LIN {X 0,Y 254.64,Z 783.41,A -85,B 0,C 180,E1 -18457.933,E2 -18457.933} C_VEL
LIN {X 0,Y 255.196,Z 782.528,A -85,B 0,C 180,E1 -18459.512,E2 -18459.512} C_VEL
LIN {X 0,Y 255.928,Z 781.105,A -85,B 0,C 180,E1 -18461.084,E2 -18461.084} C_VEL
LIN {X 0,Y 257.325,Z 777.923,A -85,B 0,C 180,E1 -18463.425,E2 -18463.425} C_VEL
LIN {X 0,Y 259.009,Z 773.292,A -85,B 0,C 180,E1 -18465.745,E2 -18465.745} C_VEL
LIN {X 0,Y 260.929,Z 768.168,A -85,B 0,C 180,E1 -18467.64,E2 -18467.64} C_VEL
LIN {X 0,Y 262.981,Z 761.785,A -85,B 0,C 180,E1 -18469.516,E2 -18469.516} C_VEL
LIN {X 0,Y 265.315,Z 753.655,A -85,B 0,C 180,E1 -18471.407,E2 -18471.407} C_VEL
LIN {X 0,Y 267.313,Z 745.611,A -85,B 0,C 180,E1 -18472.889,E2 -18472.889} C_VEL
LIN {X 0,Y 269.342,Z 736.316,A -85,B 0,C 180,E1 -18474.267,E2 -18474.267} C_VEL
LIN {X 0,Y 271.322,Z 725.43,A -85,B 0,C 180,E1 -18475.509,E2 -18475.509} C_VEL
LIN {X 0,Y 272.904,Z 714.301,A -85,B 0,C 180,E1 -18476.479,E2 -18476.479} C_VEL
LIN {X 0,Y 274.215,Z 699.395,A -85,B 0,C 180,E1 -18477.423,E2 -18477.423} C_VEL
LIN {X 0,Y 278.601,Z 663.75,A -85,B 0,C 180,E1 -18479.26,E2 -18479.26} C_VEL
LIN {X 0,Y 282.632,Z 634.038,A -85,B 0,C 180,E1 -18480.701,E2 -18480.701} C_VEL
LIN {X 0,Y 282.883,Z 631.989,A -85,B 0,C 180,E1 -18480.826,E2 -18480.826} C_VEL
LIN {X 0,Y 286.551,Z 622.135,A -85,B 0,C 180,E1 -18481.825,E2 -18481.825} C_VEL
LIN {X 0,Y 289.01,Z 614.087,A -85,B 0,C 180,E1 -18483.007,E2 -18483.007} C_VEL
LIN {X 0,Y 289.054,Z 610.102,A -85,B 0,C 180,E1 -18484.242,E2 -18484.242} C_VEL
LIN {X 0,Y 288.786,Z 608.298,A -85,B 0,C 180,E1 -18485.033,E2 -18485.033} C_VEL
LIN {X 0,Y 287.847,Z 606.637,A -85,B 0,C 180,E1 -18486.32,E2 -18486.32} C_VEL
LIN {X 0,Y 286.56,Z 604.936,A -85,B 0,C 180,E1 -18488.296,E2 -18488.296} C_VEL
LIN {X 0,Y 285.583,Z 604.023,A -85,B 0,C 180,E1 -18490.28,E2 -18490.28} C_VEL
LIN {X 0,Y 284.947,Z 603.772,A -85,B 0,C 180,E1 -18492.275,E2 -18492.275} C_VEL
LIN {X 0,Y 284.613,Z 604.193,A -85,B 0,C 180,E1 -18494.266,E2 -18494.266} C_VEL
LIN {X 0,Y 284.469,Z 605.335,A -85,B 0,C 180,E1 -18496.23,E2 -18496.23} C_VEL
LIN {X 0,Y 284.524,Z 608.104,A -85,B 0,C 180,E1 -18498.967,E2 -18498.967} C_VEL
LIN {X 0,Y 284.591,Z 611.178,A -85,B 0,C 180,E1 -18501.037,E2 -18501.037} C_VEL
LIN {X 0,Y 284.604,Z 615.38,A -85,B 0,C 180,E1 -18503.209,E2 -18503.209} C_VEL
LIN {X 0,Y 284.52,Z 617.632,A -85,B 0,C 180,E1 -18504.2,E2 -18504.2} C_VEL
LIN {X 0,Y 283.942,Z 619.835,A -85,B 0,C 180,E1 -18504.867,E2 -18504.867} C_VEL
LIN {X 0,Y 279.716,Z 632.839,A -85,B 0,C 180,E1 -18508.101,E2 -18508.101} C_VEL
LIN {X 0,Y 281.369,Z 646.293,A -85,B 0,C 180,E1 -18509.997,E2 -18509.997} C_VEL
LIN {X 0,Y 282.942,Z 661.375,A -85,B 0,C 180,E1 -18511.756,E2 -18511.756} C_VEL
LIN {X 0,Y 283.284,Z 668.767,A -85,B 0,C 180,E1 -18512.455,E2 -18512.455} C_VEL
LIN {X 0,Y 278.495,Z 708.238,A -85,B 0,C 180,E1 -18514.295,E2 -18514.295} C_VEL
LIN {X 0,Y 276.699,Z 719.034,A -85,B 0,C 180,E1 -18515.022,E2 -18515.022} C_VEL
LIN {X 0,Y 274.44,Z 729.554,A -85,B 0,C 180,E1 -18516.013,E2 -18516.013} C_VEL
LIN {X 0,Y 272.006,Z 739.288,A -85,B 0,C 180,E1 -18517.197,E2 -18517.197} C_VEL
LIN {X 0,Y 269.353,Z 748.071,A -85,B 0,C 180,E1 -18518.575,E2 -18518.575} C_VEL
LIN {X 0,Y 267,Z 755.114,A -85,B 0,C 180,E1 -18519.99,E2 -18519.99} C_VEL
LIN {X 0,Y 264.343,Z 762.314,A -85,B 0,C 180,E1 -18521.796,E2 -18521.796} C_VEL
LIN {X 0,Y 261.944,Z 768.017,A -85,B 0,C 180,E1 -18523.637,E2 -18523.637} C_VEL
LIN {X 0,Y 259.412,Z 773.188,A -85,B 0,C 180,E1 -18525.887,E2 -18525.887} C_VEL
LIN {X 0,Y 258.13,Z 775.765,A -85,B 0,C 180,E1 -18527.419,E2 -18527.419} C_VEL
LIN {X 0,Y 257.031,Z 777.741,A -85,B 0,C 180,E1 -18528.965,E2 -18528.965} C_VEL
LIN {X 0,Y 256.07,Z 779.154,A -85,B 0,C 180,E1 -18530.522,E2 -18530.522} C_VEL
LIN {X 0,Y 255.228,Z 780.071,A -85,B 0,C 180,E1 -18532.445,E2 -18532.445} C_VEL
LIN {X 0,Y 254.805,Z 780.276,A -85,B 0,C 180,E1 -18533.666,E2 -18533.666} C_VEL
LIN {X 0,Y 254.337,Z 779.949,A -85,B 0,C 180,E1 -18535.245,E2 -18535.245} C_VEL
LIN {X 0,Y 254.123,Z 779.049,A -85,B 0,C 180,E1 -18536.829,E2 -18536.829} C_VEL
LIN {X 0,Y 254.003,Z 776.68,A -85,B 0,C 180,E1 -18539.207,E2 -18539.207} C_VEL
LIN {X 0,Y 254.05,Z 772.777,A -85,B 0,C 180,E1 -18541.585,E2 -18541.585} C_VEL
LIN {X 0,Y 254.225,Z 769.338,A -85,B 0,C 180,E1 -18543.17,E2 -18543.17} C_VEL
LIN {X 0,Y 254.358,Z 765.073,A -85,B 0,C 180,E1 -18544.755,E2 -18544.755} C_VEL
LIN {X 0,Y 254.634,Z 758.449,A -85,B 0,C 180,E1 -18546.737,E2 -18546.737} C_VEL
LIN {X 0,Y 254.986,Z 751.78,A -85,B 0,C 180,E1 -18548.32,E2 -18548.32} C_VEL
LIN {X 0,Y 255.449,Z 743.401,A -85,B 0,C 180,E1 -18549.901,E2 -18549.901} C_VEL
LIN {X 0,Y 255.9,Z 734.328,A -85,B 0,C 180,E1 -18551.285,E2 -18551.285} C_VEL
LIN {X 0,Y 256.485,Z 723.294,A -85,B 0,C 180,E1 -18552.562,E2 -18552.562} C_VEL
LIN {X 0,Y 256.869,Z 713.102,A -85,B 0,C 180,E1 -18553.448,E2 -18553.448} C_VEL
LIN {X 0,Y 257.314,Z 700.732,A -85,B 0,C 180,E1 -18554.18,E2 -18554.18} C_VEL
LIN {X 0,Y 258.285,Z 654.86,A -85,B 0,C 180,E1 -18556.218,E2 -18556.218} C_VEL
LIN {X 0,Y 256.91,Z 633.005,A -85,B 0,C 180,E1 -18557.211,E2 -18557.211} C_VEL
LIN {X 0,Y 256.915,Z 631.92,A -85,B 0,C 180,E1 -18557.311,E2 -18557.311} C_VEL
LIN {X 0,Y 258.388,Z 612.535,A -85,B 0,C 180,E1 -18561.543,E2 -18561.543} C_VEL
LIN {X 0,Y 259.975,Z 593.835,A -85,B 0,C 180,E1 -18565.629,E2 -18565.629} C_VEL
LIN {X 0,Y 261.374,Z 578.642,A -85,B 0,C 180,E1 -18568.947,E2 -18568.947} C_VEL
LIN {X 0,Y 260.158,Z 571.5,A -85,B 0,C 180,E1 -18570.601,E2 -18570.601} C_VEL
LIN {X 0,Y 256.188,Z 552.77,A -85,B 0,C 180,E1 -18575.125,E2 -18575.125} C_VEL
LIN {X 0,Y 256.077,Z 552.583,A -85,B 0,C 180,E1 -18579.141,E2 -18579.141} C_VEL
LIN {X 0,Y 256.07,Z 552.534,A -85,B 0,C 180,E1 -18583.326,E2 -18583.326} C_VEL
LIN {X 0,Y 256.093,Z 552.578,A -85,B 0,C 180,E1 -18587.814,E2 -18587.814} C_VEL
LIN {X 0,Y 256.078,Z 552.55,A -85,B 0,C 180,E1 -18590.858,E2 -18590.858} C_VEL
LIN {X 0,Y 256.134,Z 552.571,A -85,B 0,C 180,E1 -18592.867,E2 -18592.867} C_VEL
LIN {X 0,Y 256.153,Z 552.697,A -85,B 0,C 180,E1 -18596.5,E2 -18596.5} C_VEL
LIN {X 0,Y 256.89,Z 555.634,A -85,B 0,C 180,E1 -18597.795,E2 -18597.795} C_VEL
LIN {X 0,Y 264.799,Z 571.908,A -85,B 0,C 180,E1 -18599.433,E2 -18599.433} C_VEL
LIN {X 0,Y 271.817,Z 588.537,A -85,B 0,C 180,E1 -18600.806,E2 -18600.806} C_VEL
LIN {X 0,Y 273.608,Z 593.478,A -85,B 0,C 180,E1 -18601.163,E2 -18601.163} C_VEL
LIN {X 0,Y 271.526,Z 660.332,A -85,B 0,C 180,E1 -18602.909,E2 -18602.909} C_VEL
LIN {X 0,Y 270.584,Z 673.573,A -85,B 0,C 180,E1 -18603.485,E2 -18603.485} C_VEL
LIN {X 0,Y 269.339,Z 686.707,A -85,B 0,C 180,E1 -18604.393,E2 -18604.393} C_VEL
LIN {X 0,Y 267.637,Z 699.141,A -85,B 0,C 180,E1 -18605.568,E2 -18605.568} C_VEL
LIN {X 0,Y 265.652,Z 710.78,A -85,B 0,C 180,E1 -18607.03,E2 -18607.03} C_VEL
LIN {X 0,Y 263.919,Z 719.999,A -85,B 0,C 180,E1 -18608.488,E2 -18608.488} C_VEL
LIN {X 0,Y 262.043,Z 729.759,A -85,B 0,C 180,E1 -18610.411,E2 -18610.411} C_VEL
LIN {X 0,Y 260.236,Z 737.623,A -85,B 0,C 180,E1 -18612.311,E2 -18612.311} C_VEL
LIN {X 0,Y 258.368,Z 745.305,A -85,B 0,C 180,E1 -18614.619,E2 -18614.619} C_VEL
LIN {X 0,Y 256.723,Z 752.357,A -85,B 0,C 180,E1 -18617.348,E2 -18617.348} C_VEL
LIN {X 0,Y 255.59,Z 757.052,A -85,B 0,C 180,E1 -18619.703,E2 -18619.703} C_VEL
LIN {X 0,Y 254.885,Z 760.637,A -85,B 0,C 180,E1 -18622.074,E2 -18622.074} C_VEL
LIN {X 0,Y 254.515,Z 762.597,A -85,B 0,C 180,E1 -18623.765,E2 -18623.765} C_VEL
LIN {X 0,Y 254.194,Z 764.873,A -85,B 0,C 180,E1 -18626.829,E2 -18626.829} C_VEL
LIN {X 0,Y 254.096,Z 765.484,A -85,B 0,C 180,E1 -18628.414,E2 -18628.414} C_VEL
LIN {X 0,Y 254.064,Z 765.714,A -85,B 0,C 180,E1 -18629.999,E2 -18629.999} C_VEL
LIN {X 0,Y 254.095,Z 765.522,A -85,B 0,C 180,E1 -18631.584,E2 -18631.584} C_VEL
LIN {X 0,Y 254.192,Z 764.937,A -85,B 0,C 180,E1 -18633.168,E2 -18633.168} C_VEL
LIN {X 0,Y 254.534,Z 762.617,A -85,B 0,C 180,E1 -18636.339,E2 -18636.339} C_VEL
LIN {X 0,Y 255.077,Z 759.749,A -85,B 0,C 180,E1 -18638.715,E2 -18638.715} C_VEL
LIN {X 0,Y 255.91,Z 755.858,A -85,B 0,C 180,E1 -18641.082,E2 -18641.082} C_VEL
LIN {X 0,Y 257.1,Z 750.84,A -85,B 0,C 180,E1 -18643.434,E2 -18643.434} C_VEL
LIN {X 0,Y 258.531,Z 744.522,A -85,B 0,C 180,E1 -18645.772,E2 -18645.772} C_VEL
LIN {X 0,Y 260.488,Z 736.605,A -85,B 0,C 180,E1 -18648.074,E2 -18648.074} C_VEL
LIN {X 0,Y 262.351,Z 728.536,A -85,B 0,C 180,E1 -18649.97,E2 -18649.97} C_VEL
LIN {X 0,Y 264.206,Z 718.694,A -85,B 0,C 180,E1 -18651.862,E2 -18651.862} C_VEL
LIN {X 0,Y 266.253,Z 707.61,A -85,B 0,C 180,E1 -18653.529,E2 -18653.529} C_VEL
LIN {X 0,Y 268.044,Z 696.735,A -85,B 0,C 180,E1 -18654.802,E2 -18654.802} C_VEL
LIN {X 0,Y 269.616,Z 684.708,A -85,B 0,C 180,E1 -18655.887,E2 -18655.887} C_VEL
LIN {X 0,Y 270.803,Z 672.349,A -85,B 0,C 180,E1 -18656.697,E2 -18656.697} C_VEL
LIN {X 0,Y 271.68,Z 659.521,A -85,B 0,C 180,E1 -18657.228,E2 -18657.228} C_VEL
LIN {X 0,Y 273.728,Z 593.612,A -85,B 0,C 180,E1 -18658.945,E2 -18658.945} C_VEL
LIN {X 0,Y 266.65,Z 575.933,A -85,B 0,C 180,E1 -18660.336,E2 -18660.336} C_VEL
LIN {X 0,Y 258.473,Z 559.011,A -85,B 0,C 180,E1 -18661.953,E2 -18661.953} C_VEL
LIN {X 0,Y 256.796,Z 555.428,A -85,B 0,C 180,E1 -18662.39,E2 -18662.39} C_VEL
LIN {X 0,Y 256.138,Z 552.622,A -85,B 0,C 180,E1 -18663.719,E2 -18663.719} C_VEL
LIN {X 0,Y 256.127,Z 552.578,A -85,B 0,C 180,E1 -18667.274,E2 -18667.274} C_VEL
LIN {X 0,Y 256.053,Z 552.584,A -85,B 0,C 180,E1 -18671.201,E2 -18671.201} C_VEL
LIN {X 0,Y 256.057,Z 552.569,A -85,B 0,C 180,E1 -18675.528,E2 -18675.528} C_VEL
LIN {X 0,Y 256.079,Z 552.582,A -85,B 0,C 180,E1 -18678.801,E2 -18678.801} C_VEL
LIN {X 0,Y 256.149,Z 552.557,A -85,B 0,C 180,E1 -18682.87,E2 -18682.87} C_VEL
LIN {X 0,Y 256.08,Z 552.582,A -85,B 0,C 180,E1 -18686.709,E2 -18686.709} C_VEL
LIN {X 0,Y 256.132,Z 552.572,A -85,B 0,C 180,E1 -18691.404,E2 -18691.404} C_VEL
LIN {X 0,Y 256.149,Z 552.574,A -85,B 0,C 180,E1 -18695.822,E2 -18695.822} C_VEL
LIN {X 0,Y 256.16,Z 552.567,A -85,B 0,C 180,E1 -18699.104,E2 -18699.104} C_VEL
LIN {X 0,Y 256.208,Z 552.56,A -85,B 0,C 180,E1 -18702.664,E2 -18702.664} C_VEL
LIN {X 0,Y 255.561,Z 552.637,A -85,B 0,C 180,E1 -18703.976,E2 -18703.976} C_VEL
LIN {X 0,Y 252.702,Z 553.006,A -85,B 0,C 180,E1 -18706.116,E2 -18706.116} C_VEL
LIN {X 0,Y 250.308,Z 553.301,A -85,B 0,C 180,E1 -18707.859,E2 -18707.859} C_VEL
LIN {X 0,Y 249.349,Z 553.411,A -85,B 0,C 180,E1 -18709.21,E2 -18709.21} C_VEL
LIN {X 0,Y 249.309,Z 553.412,A -85,B 0,C 180,E1 -18709.667,E2 -18709.667} C_VEL
LIN {X 0,Y 249.475,Z 553.401,A -85,B 0,C 180,E1 -18711.903,E2 -18711.903} C_VEL
LIN {X 0,Y 249.43,Z 553.396,A -85,B 0,C 180,E1 -18716.769,E2 -18716.769} C_VEL
LIN {X 0,Y 249.729,Z 553.378,A -85,B 0,C 180,E1 -18720,E2 -18720} C_VEL
LIN {X 0,Y 249.43,Z 553.398,A -85,B 0,C 180,E1 -18723.23,E2 -18723.23} C_VEL
LIN {X 0,Y 249.478,Z 553.404,A -85,B 0,C 180,E1 -18728.097,E2 -18728.097} C_VEL
LIN {X 0,Y 249.246,Z 553.426,A -85,B 0,C 180,E1 -18731.384,E2 -18731.384} C_VEL
LIN {X 0,Y 249.235,Z 553.424,A -85,B 0,C 180,E1 -18736.379,E2 -18736.379} C_VEL
LIN {X 0,Y 249.081,Z 553.447,A -85,B 0,C 180,E1 -18741.519,E2 -18741.519} C_VEL
LIN {X 0,Y 249.123,Z 553.448,A -85,B 0,C 180,E1 -18745.482,E2 -18745.482} C_VEL
LIN {X 0,Y 249.066,Z 553.461,A -85,B 0,C 180,E1 -18748.99,E2 -18748.99} C_VEL
LIN {X 0,Y 249.024,Z 553.465,A -85,B 0,C 180,E1 -18752.427,E2 -18752.427} C_VEL
LIN {X 0,Y 249.024,Z 553.436,A -85,B 0,C 180,E1 -18756.346,E2 -18756.346} C_VEL
LIN {X 0,Y 249.03,Z 553.464,A -85,B 0,C 180,E1 -18760.473,E2 -18760.473} C_VEL
LIN {X 0,Y 249.015,Z 553.468,A -85,B 0,C 180,E1 -18764.877,E2 -18764.877} C_VEL
LIN {X 0,Y 249.077,Z 553.446,A -85,B 0,C 180,E1 -18767.378,E2 -18767.378} C_VEL
LIN {X 0,Y 249.119,Z 553.651,A -85,B 0,C 180,E1 -18771.056,E2 -18771.056} C_VEL
LIN {X 0,Y 250.889,Z 560.889,A -85,B 0,C 180,E1 -18774.327,E2 -18774.327} C_VEL
LIN {X 0,Y 252.417,Z 567.594,A -85,B 0,C 180,E1 -18777.053,E2 -18777.053} C_VEL
LIN {X 0,Y 258.204,Z 580.32,A -85,B 0,C 180,E1 -18778.332,E2 -18778.332} C_VEL
LIN {X 0,Y 263,Z 592.075,A -85,B 0,C 180,E1 -18779.336,E2 -18779.336} C_VEL
LIN {X 0,Y 266.778,Z 617.218,A -85,B 0,C 180,E1 -18780.575,E2 -18780.575} C_VEL
LIN {X 0,Y 264.813,Z 676.163,A -85,B 0,C 180,E1 -18782.167,E2 -18782.167} C_VEL
LIN {X 0,Y 263.611,Z 690.053,A -85,B 0,C 180,E1 -18782.836,E2 -18782.836} C_VEL
LIN {X 0,Y 262.061,Z 702.494,A -85,B 0,C 180,E1 -18783.738,E2 -18783.738} C_VEL
LIN {X 0,Y 260.345,Z 713.602,A -85,B 0,C 180,E1 -18784.84,E2 -18784.84} C_VEL
LIN {X 0,Y 258.166,Z 725.168,A -85,B 0,C 180,E1 -18786.327,E2 -18786.327} C_VEL
LIN {X 0,Y 255.993,Z 735.585,A -85,B 0,C 180,E1 -18788.036,E2 -18788.036} C_VEL
LIN {X 0,Y 254.117,Z 744.109,A -85,B 0,C 180,E1 -18789.777,E2 -18789.777} C_VEL
LIN {X 0,Y 252.362,Z 752.159,A -85,B 0,C 180,E1 -18791.797,E2 -18791.797} C_VEL
LIN {X 0,Y 250.528,Z 759.66,A -85,B 0,C 180,E1 -18794.128,E2 -18794.128} C_VEL
LIN {X 0,Y 248.79,Z 766.747,A -85,B 0,C 180,E1 -18796.94,E2 -18796.94} C_VEL
LIN {X 0,Y 247.858,Z 771.468,A -85,B 0,C 180,E1 -18799.381,E2 -18799.381} C_VEL
LIN {X 0,Y 247.267,Z 775.082,A -85,B 0,C 180,E1 -18801.831,E2 -18801.831} C_VEL
LIN {X 0,Y 247.009,Z 776.944,A -85,B 0,C 180,E1 -18803.467,E2 -18803.467} C_VEL
LIN {X 0,Y 246.882,Z 778.341,A -85,B 0,C 180,E1 -18805.102,E2 -18805.102} C_VEL
LIN {X 0,Y 246.865,Z 779.339,A -85,B 0,C 180,E1 -18806.737,E2 -18806.737} C_VEL
LIN {X 0,Y 246.923,Z 779.949,A -85,B 0,C 180,E1 -18808.37,E2 -18808.37} C_VEL
LIN {X 0,Y 246.949,Z 780.095,A -85,B 0,C 180,E1 -18811.225,E2 -18811.225} C_VEL
LIN {X 0,Y 246.947,Z 782.169,A -85,B 0,C 180,E1 -18813.264,E2 -18813.264} C_VEL
LIN {X 0,Y 247.047,Z 783.354,A -85,B 0,C 180,E1 -18815.325,E2 -18815.325} C_VEL
LIN {X 0,Y 247.614,Z 783.463,A -85,B 0,C 180,E1 -18818.16,E2 -18818.16} C_VEL
LIN {X 0,Y 248.201,Z 782.811,A -85,B 0,C 180,E1 -18819.783,E2 -18819.783} C_VEL
LIN {X 0,Y 248.985,Z 781.614,A -85,B 0,C 180,E1 -18821.397,E2 -18821.397} C_VEL
LIN {X 0,Y 250.463,Z 778.708,A -85,B 0,C 180,E1 -18823.8,E2 -18823.8} C_VEL
LIN {X 0,Y 252.303,Z 774.521,A -85,B 0,C 180,E1 -18826.175,E2 -18826.175} C_VEL
LIN {X 0,Y 254.75,Z 768.662,A -85,B 0,C 180,E1 -18828.499,E2 -18828.499} C_VEL
LIN {X 0,Y 257.017,Z 762.49,A -85,B 0,C 180,E1 -18830.406,E2 -18830.406} C_VEL
LIN {X 0,Y 259.535,Z 754.826,A -85,B 0,C 180,E1 -18832.28,E2 -18832.28} C_VEL
LIN {X 0,Y 262.002,Z 746.136,A -85,B 0,C 180,E1 -18833.938,E2 -18833.938} C_VEL
LIN {X 0,Y 264.356,Z 736.691,A -85,B 0,C 180,E1 -18835.386,E2 -18835.386} C_VEL
LIN {X 0,Y 266.514,Z 725.928,A -85,B 0,C 180,E1 -18836.635,E2 -18836.635} C_VEL
LIN {X 0,Y 268.425,Z 714.14,A -85,B 0,C 180,E1 -18837.694,E2 -18837.694} C_VEL
LIN {X 0,Y 270.241,Z 697.254,A -85,B 0,C 180,E1 -18838.76,E2 -18838.76} C_VEL
LIN {X 0,Y 274.782,Z 663.805,A -85,B 0,C 180,E1 -18840.501,E2 -18840.501} C_VEL
LIN {X 0,Y 279.106,Z 634.046,A -85,B 0,C 180,E1 -18841.978,E2 -18841.978} C_VEL
LIN {X 0,Y 279.349,Z 632.11,A -85,B 0,C 180,E1 -18842.106,E2 -18842.106} C_VEL
LIN {X 0,Y 282.562,Z 623.941,A -85,B 0,C 180,E1 -18842.963,E2 -18842.963} C_VEL
LIN {X 0,Y 284.56,Z 618.001,A -85,B 0,C 180,E1 -18843.841,E2 -18843.841} C_VEL
LIN {X 0,Y 284.694,Z 615.564,A -85,B 0,C 180,E1 -18844.597,E2 -18844.597} C_VEL
LIN {X 0,Y 284.501,Z 613.728,A -85,B 0,C 180,E1 -18845.393,E2 -18845.393} C_VEL
LIN {X 0,Y 283.058,Z 611.491,A -85,B 0,C 180,E1 -18847.39,E2 -18847.39} C_VEL
LIN {X 0,Y 281.903,Z 610.195,A -85,B 0,C 180,E1 -18849.39,E2 -18849.39} C_VEL
LIN {X 0,Y 281.036,Z 609.577,A -85,B 0,C 180,E1 -18851.39,E2 -18851.39} C_VEL
LIN {X 0,Y 280.49,Z 609.675,A -85,B 0,C 180,E1 -18853.395,E2 -18853.395} C_VEL
LIN {X 0,Y 280.182,Z 610.456,A -85,B 0,C 180,E1 -18855.385,E2 -18855.385} C_VEL
LIN {X 0,Y 280.014,Z 611.963,A -85,B 0,C 180,E1 -18857.338,E2 -18857.338} C_VEL
LIN {X 0,Y 279.951,Z 614.125,A -85,B 0,C 180,E1 -18859.253,E2 -18859.253} C_VEL
LIN {X 0,Y 279.836,Z 618.383,A -85,B 0,C 180,E1 -18861.924,E2 -18861.924} C_VEL
LIN {X 0,Y 279.619,Z 621.758,A -85,B 0,C 180,E1 -18863.544,E2 -18863.544} C_VEL
LIN {X 0,Y 278.918,Z 624.069,A -85,B 0,C 180,E1 -18864.26,E2 -18864.26} C_VEL
LIN {X 0,Y 275.821,Z 633.078,A -85,B 0,C 180,E1 -18866.523,E2 -18866.523} C_VEL
LIN {X 0,Y 277.151,Z 646.617,A -85,B 0,C 180,E1 -18868.591,E2 -18868.591} C_VEL
LIN {X 0,Y 278.438,Z 661.312,A -85,B 0,C 180,E1 -18870.437,E2 -18870.437} C_VEL
LIN {X 0,Y 278.893,Z 670.399,A -85,B 0,C 180,E1 -18871.362,E2 -18871.362} C_VEL
LIN {X 0,Y 273.775,Z 708.71,A -85,B 0,C 180,E1 -18873.202,E2 -18873.202} C_VEL
LIN {X 0,Y 271.883,Z 719.441,A -85,B 0,C 180,E1 -18873.932,E2 -18873.932} C_VEL
LIN {X 0,Y 269.494,Z 729.878,A -85,B 0,C 180,E1 -18874.927,E2 -18874.927} C_VEL
LIN {X 0,Y 266.898,Z 739.436,A -85,B 0,C 180,E1 -18876.118,E2 -18876.118} C_VEL
LIN {X 0,Y 263.7,Z 749.041,A -85,B 0,C 180,E1 -18877.68,E2 -18877.68} C_VEL
LIN {X 0,Y 261.19,Z 755.969,A -85,B 0,C 180,E1 -18879.113,E2 -18879.113} C_VEL
LIN {X 0,Y 258.353,Z 763.027,A -85,B 0,C 180,E1 -18880.947,E2 -18880.947} C_VEL
LIN {X 0,Y 256.218,Z 767.56,A -85,B 0,C 180,E1 -18882.439,E2 -18882.439} C_VEL
LIN {X 0,Y 253.458,Z 772.814,A -85,B 0,C 180,E1 -18884.727,E2 -18884.727} C_VEL
LIN {X 0,Y 251.953,Z 775.512,A -85,B 0,C 180,E1 -18886.285,E2 -18886.285} C_VEL
LIN {X 0,Y 250.12,Z 778.385,A -85,B 0,C 180,E1 -18888.657,E2 -18888.657} C_VEL
LIN {X 0,Y 249.095,Z 779.553,A -85,B 0,C 180,E1 -18890.254,E2 -18890.254} C_VEL
LIN {X 0,Y 248.077,Z 780.304,A -85,B 0,C 180,E1 -18892.552,E2 -18892.552} C_VEL
LIN {X 0,Y 247.27,Z 779.799,A -85,B 0,C 180,E1 -18895.109,E2 -18895.109} C_VEL
LIN {X 0,Y 247.049,Z 778.756,A -85,B 0,C 180,E1 -18896.738,E2 -18896.738} C_VEL
LIN {X 0,Y 246.936,Z 776.027,A -85,B 0,C 180,E1 -18899.185,E2 -18899.185} C_VEL
LIN {X 0,Y 246.993,Z 771.894,A -85,B 0,C 180,E1 -18901.631,E2 -18901.631} C_VEL
LIN {X 0,Y 247.289,Z 766.085,A -85,B 0,C 180,E1 -18904.074,E2 -18904.074} C_VEL
LIN {X 0,Y 247.439,Z 760.19,A -85,B 0,C 180,E1 -18905.953,E2 -18905.953} C_VEL
LIN {X 0,Y 247.847,Z 753.273,A -85,B 0,C 180,E1 -18907.741,E2 -18907.741} C_VEL
LIN {X 0,Y 248.337,Z 744.265,A -85,B 0,C 180,E1 -18909.571,E2 -18909.571} C_VEL
LIN {X 0,Y 248.758,Z 735.417,A -85,B 0,C 180,E1 -18910.994,E2 -18910.994} C_VEL
LIN {X 0,Y 249.293,Z 725.95,A -85,B 0,C 180,E1 -18912.207,E2 -18912.207} C_VEL
LIN {X 0,Y 249.669,Z 716.479,A -85,B 0,C 180,E1 -18913.118,E2 -18913.118} C_VEL
LIN {X 0,Y 250.074,Z 705.044,A -85,B 0,C 180,E1 -18913.924,E2 -18913.924} C_VEL
LIN {X 0,Y 251.274,Z 655.843,A -85,B 0,C 180,E1 -18916.216,E2 -18916.216} C_VEL
LIN {X 0,Y 249.82,Z 634.171,A -85,B 0,C 180,E1 -18917.225,E2 -18917.225} C_VEL
LIN {X 0,Y 249.862,Z 631.735,A -85,B 0,C 180,E1 -18917.432,E2 -18917.432} C_VEL
LIN {X 0,Y 251.202,Z 614.313,A -85,B 0,C 180,E1 -18921.328,E2 -18921.328} C_VEL
LIN {X 0,Y 252.809,Z 595.512,A -85,B 0,C 180,E1 -18925.525,E2 -18925.525} C_VEL
LIN {X 0,Y 254.351,Z 579.257,A -85,B 0,C 180,E1 -18929.144,E2 -18929.144} C_VEL
LIN {X 0,Y 252.358,Z 568.974,A -85,B 0,C 180,E1 -18931.591,E2 -18931.591} C_VEL
LIN {X 0,Y 249.166,Z 553.642,A -85,B 0,C 180,E1 -18935.393,E2 -18935.393} C_VEL
LIN {X 0,Y 249.031,Z 553.466,A -85,B 0,C 180,E1 -18938.38,E2 -18938.38} C_VEL
LIN {X 0,Y 249.016,Z 553.411,A -85,B 0,C 180,E1 -18942.792,E2 -18942.792} C_VEL
LIN {X 0,Y 249.042,Z 553.463,A -85,B 0,C 180,E1 -18947.367,E2 -18947.367} C_VEL
LIN {X 0,Y 249.031,Z 553.433,A -85,B 0,C 180,E1 -18951.619,E2 -18951.619} C_VEL
LIN {X 0,Y 249.067,Z 553.51,A -85,B 0,C 180,E1 -18955.642,E2 -18955.642} C_VEL
LIN {X 0,Y 249.562,Z 555.442,A -85,B 0,C 180,E1 -18956.621,E2 -18956.621} C_VEL
LIN {X 0,Y 250.069,Z 556.882,A -85,B 0,C 180,E1 -18956.882,E2 -18956.882} C_VEL
LIN {X 0,Y 257.895,Z 572.413,A -85,B 0,C 180,E1 -18958.531,E2 -18958.531} C_VEL
LIN {X 0,Y 263.958,Z 586.258,A -85,B 0,C 180,E1 -18959.769,E2 -18959.769} C_VEL
LIN {X 0,Y 267.471,Z 595.847,A -85,B 0,C 180,E1 -18960.501,E2 -18960.501} C_VEL
LIN {X 0,Y 265.145,Z 661.962,A -85,B 0,C 180,E1 -18962.255,E2 -18962.255} C_VEL
LIN {X 0,Y 264.141,Z 675.309,A -85,B 0,C 180,E1 -18962.892,E2 -18962.892} C_VEL
LIN {X 0,Y 262.797,Z 688.047,A -85,B 0,C 180,E1 -18963.814,E2 -18963.814} C_VEL
LIN {X 0,Y 261.202,Z 699.351,A -85,B 0,C 180,E1 -18964.926,E2 -18964.926} C_VEL
LIN {X 0,Y 259.15,Z 710.988,A -85,B 0,C 180,E1 -18966.42,E2 -18966.42} C_VEL
LIN {X 0,Y 257.077,Z 721.434,A -85,B 0,C 180,E1 -18968.129,E2 -18968.129} C_VEL
LIN {X 0,Y 255.36,Z 729.966,A -85,B 0,C 180,E1 -18969.876,E2 -18969.876} C_VEL
LIN {X 0,Y 253.487,Z 737.83,A -85,B 0,C 180,E1 -18971.824,E2 -18971.824} C_VEL
LIN {X 0,Y 251.503,Z 745.513,A -85,B 0,C 180,E1 -18974.188,E2 -18974.188} C_VEL
LIN {X 0,Y 250.256,Z 750.755,A -85,B 0,C 180,E1 -18976.188,E2 -18976.188} C_VEL
LIN {X 0,Y 248.951,Z 755.843,A -85,B 0,C 180,E1 -18978.601,E2 -18978.601} C_VEL
LIN {X 0,Y 248.068,Z 759.785,A -85,B 0,C 180,E1 -18981.034,E2 -18981.034} C_VEL
LIN {X 0,Y 247.424,Z 763.002,A -85,B 0,C 180,E1 -18983.81,E2 -18983.81} C_VEL
LIN {X 0,Y 247.114,Z 765.078,A -85,B 0,C 180,E1 -18986.738,E2 -18986.738} C_VEL
LIN {X 0,Y 246.993,Z 765.918,A -85,B 0,C 180,E1 -18989.999,E2 -18989.999} C_VEL
LIN {X 0,Y 247.006,Z 765.726,A -85,B 0,C 180,E1 -18991.629,E2 -18991.629} C_VEL
LIN {X 0,Y 247.111,Z 765.141,A -85,B 0,C 180,E1 -18993.259,E2 -18993.259} C_VEL
LIN {X 0,Y 247.495,Z 762.821,A -85,B 0,C 180,E1 -18996.521,E2 -18996.521} C_VEL
LIN {X 0,Y 248.066,Z 759.953,A -85,B 0,C 180,E1 -18998.963,E2 -18998.963} C_VEL
LIN {X 0,Y 248.929,Z 756.062,A -85,B 0,C 180,E1 -19001.397,E2 -19001.397} C_VEL
LIN {X 0,Y 250.184,Z 751.044,A -85,B 0,C 180,E1 -19003.813,E2 -19003.813} C_VEL
LIN {X 0,Y 251.703,Z 744.725,A -85,B 0,C 180,E1 -19006.212,E2 -19006.212} C_VEL
LIN {X 0,Y 253.758,Z 736.807,A -85,B 0,C 180,E1 -19008.571,E2 -19008.571} C_VEL
LIN {X 0,Y 255.68,Z 728.738,A -85,B 0,C 180,E1 -19010.514,E2 -19010.514} C_VEL
LIN {X 0,Y 257.629,Z 718.895,A -85,B 0,C 180,E1 -19012.451,E2 -19012.451} C_VEL
LIN {X 0,Y 259.768,Z 707.81,A -85,B 0,C 180,E1 -19014.153,E2 -19014.153} C_VEL
LIN {X 0,Y 261.629,Z 696.933,A -85,B 0,C 180,E1 -19015.453,E2 -19015.453} C_VEL
LIN {X 0,Y 263.26,Z 684.905,A -85,B 0,C 180,E1 -19016.56,E2 -19016.56} C_VEL
LIN {X 0,Y 264.504,Z 672.541,A -85,B 0,C 180,E1 -19017.385,E2 -19017.385} C_VEL
LIN {X 0,Y 265.403,Z 659.705,A -85,B 0,C 180,E1 -19017.927,E2 -19017.927} C_VEL
LIN {X 0,Y 267.425,Z 595.252,A -85,B 0,C 180,E1 -19019.651,E2 -19019.651} C_VEL
LIN {X 0,Y 260.981,Z 579.132,A -85,B 0,C 180,E1 -19020.972,E2 -19020.972} C_VEL
LIN {X 0,Y 253.284,Z 563.062,A -85,B 0,C 180,E1 -19022.559,E2 -19022.559} C_VEL
LIN {X 0,Y 249.649,Z 555.829,A -85,B 0,C 180,E1 -19023.404,E2 -19023.404} C_VEL
LIN {X 0,Y 249.109,Z 553.695,A -85,B 0,C 180,E1 -19024.348,E2 -19024.348} C_VEL
LIN {X 0,Y 249.067,Z 553.451,A -85,B 0,C 180,E1 -19026.337,E2 -19026.337} C_VEL
LIN {X 0,Y 249.022,Z 553.452,A -85,B 0,C 180,E1 -19030.473,E2 -19030.473} C_VEL
LIN {X 0,Y 249,Z 553.446,A -85,B 0,C 180,E1 -19034.877,E2 -19034.877} C_VEL
LIN {X 0,Y 249.023,Z 553.464,A -85,B 0,C 180,E1 -19037.364,E2 -19037.364} C_VEL
LIN {X 0,Y 249.046,Z 553.431,A -85,B 0,C 180,E1 -19041.623,E2 -19041.623} C_VEL
LIN {X 0,Y 249.057,Z 553.463,A -85,B 0,C 180,E1 -19045.641,E2 -19045.641} C_VEL
LIN {X 0,Y 249.046,Z 553.463,A -85,B 0,C 180,E1 -19049.472,E2 -19049.472} C_VEL
LIN {X 0,Y 249.068,Z 553.449,A -85,B 0,C 180,E1 -19053.161,E2 -19053.161} C_VEL
LIN {X 0,Y 249.073,Z 553.451,A -85,B 0,C 180,E1 -19056.732,E2 -19056.732} C_VEL
LIN {X 0,Y 249.105,Z 553.454,A -85,B 0,C 180,E1 -19060.211,E2 -19060.211} C_VEL
LIN {X 0,Y 249.235,Z 553.422,A -85,B 0,C 180,E1 -19063.621,E2 -19063.621} C_VEL
LIN {X 0,Y 249.246,Z 553.43,A -85,B 0,C 180,E1 -19068.616,E2 -19068.616} C_VEL
LIN {X 0,Y 249.309,Z 553.412,A -85,B 0,C 180,E1 -19069.667,E2 -19069.667} C_VEL
LIN {X 0,Y 248.722,Z 553.488,A -85,B 0,C 180,E1 -19071.016,E2 -19071.016} C_VEL
LIN {X 0,Y 245.848,Z 553.861,A -85,B 0,C 180,E1 -19073.213,E2 -19073.213} C_VEL
LIN {X 0,Y 243.403,Z 554.16,A -85,B 0,C 180,E1 -19075.004,E2 -19075.004} C_VEL
LIN {X 0,Y 242.425,Z 554.27,A -85,B 0,C 180,E1 -19076.394,E2 -19076.394} C_VEL
LIN {X 0,Y 242.388,Z 554.273,A -85,B 0,C 180,E1 -19076.865,E2 -19076.865} C_VEL
LIN {X 0,Y 242.692,Z 554.255,A -85,B 0,C 180,E1 -19080,E2 -19080} C_VEL
LIN {X 0,Y 242.631,Z 554.256,A -85,B 0,C 180,E1 -19081.66,E2 -19081.66} C_VEL
LIN {X 0,Y 242.428,Z 554.286,A -85,B 0,C 180,E1 -19086.659,E2 -19086.659} C_VEL
LIN {X 0,Y 242.339,Z 554.28,A -85,B 0,C 180,E1 -19090.021,E2 -19090.021} C_VEL
LIN {X 0,Y 242.16,Z 554.31,A -85,B 0,C 180,E1 -19095.141,E2 -19095.141} C_VEL
LIN {X 0,Y 242.067,Z 554.331,A -85,B 0,C 180,E1 -19098.625,E2 -19098.625} C_VEL
LIN {X 0,Y 242.007,Z 554.328,A -85,B 0,C 180,E1 -19102.181,E2 -19102.181} C_VEL
LIN {X 0,Y 242.06,Z 554.324,A -85,B 0,C 180,E1 -19105.839,E2 -19105.839} C_VEL
LIN {X 0,Y 242.001,Z 554.339,A -85,B 0,C 180,E1 -19109.584,E2 -19109.584} C_VEL
LIN {X 0,Y 241.975,Z 554.344,A -85,B 0,C 180,E1 -19113.494,E2 -19113.494} C_VEL
LIN {X 0,Y 241.985,Z 554.317,A -85,B 0,C 180,E1 -19117.583,E2 -19117.583} C_VEL
LIN {X 0,Y 241.95,Z 554.328,A -85,B 0,C 180,E1 -19121.92,E2 -19121.92} C_VEL
LIN {X 0,Y 241.998,Z 554.328,A -85,B 0,C 180,E1 -19126.556,E2 -19126.556} C_VEL
LIN {X 0,Y 242.066,Z 554.398,A -85,B 0,C 180,E1 -19130.063,E2 -19130.063} C_VEL
LIN {X 0,Y 243.966,Z 562.141,A -85,B 0,C 180,E1 -19133.766,E2 -19133.766} C_VEL
LIN {X 0,Y 245.178,Z 567.219,A -85,B 0,C 180,E1 -19135.926,E2 -19135.926} C_VEL
LIN {X 0,Y 248.049,Z 573.649,A -85,B 0,C 180,E1 -19136.659,E2 -19136.659} C_VEL
LIN {X 0,Y 254.453,Z 587.838,A -85,B 0,C 180,E1 -19138.058,E2 -19138.058} C_VEL
LIN {X 0,Y 257.269,Z 595.435,A -85,B 0,C 180,E1 -19138.689,E2 -19138.689} C_VEL
LIN {X 0,Y 260.627,Z 618.503,A -85,B 0,C 180,E1 -19139.855,E2 -19139.855} C_VEL
LIN {X 0,Y 258.556,Z 675.972,A -85,B 0,C 180,E1 -19141.432,E2 -19141.432} C_VEL
LIN {X 0,Y 257.328,Z 689.858,A -85,B 0,C 180,E1 -19142.116,E2 -19142.116} C_VEL
LIN {X 0,Y 255.692,Z 702.295,A -85,B 0,C 180,E1 -19143.032,E2 -19143.032} C_VEL
LIN {X 0,Y 253.642,Z 714.986,A -85,B 0,C 180,E1 -19144.347,E2 -19144.347} C_VEL
LIN {X 0,Y 251.396,Z 726.26,A -85,B 0,C 180,E1 -19145.869,E2 -19145.869} C_VEL
LIN {X 0,Y 249.155,Z 736.42,A -85,B 0,C 180,E1 -19147.619,E2 -19147.619} C_VEL
LIN {X 0,Y 247.055,Z 745.579,A -85,B 0,C 180,E1 -19149.608,E2 -19149.608} C_VEL
LIN {X 0,Y 245.288,Z 753.149,A -85,B 0,C 180,E1 -19151.63,E2 -19151.63} C_VEL
LIN {X 0,Y 243.378,Z 760.577,A -85,B 0,C 180,E1 -19154.08,E2 -19154.08} C_VEL
LIN {X 0,Y 241.836,Z 766.542,A -85,B 0,C 180,E1 -19156.558,E2 -19156.558} C_VEL
LIN {X 0,Y 240.859,Z 771.264,A -85,B 0,C 180,E1 -19159.068,E2 -19159.068} C_VEL
LIN {X 0,Y 240.214,Z 774.877,A -85,B 0,C 180,E1 -19161.59,E2 -19161.59} C_VEL
LIN {X 0,Y 239.951,Z 776.74,A -85,B 0,C 180,E1 -19163.274,E2 -19163.274} C_VEL
LIN {X 0,Y 239.773,Z 778.339,A -85,B 0,C 180,E1 -19165.258,E2 -19165.258} C_VEL
LIN {X 0,Y 239.833,Z 779.744,A -85,B 0,C 180,E1 -19168.322,E2 -19168.322} C_VEL
LIN {X 0,Y 239.864,Z 779.838,A -85,B 0,C 180,E1 -19171.261,E2 -19171.261} C_VEL
LIN {X 0,Y 239.901,Z 779.824,A -85,B 0,C 180,E1 -19171.68,E2 -19171.68} C_VEL
LIN {X 0,Y 239.895,Z 781.571,A -85,B 0,C 180,E1 -19173.361,E2 -19173.361} C_VEL
LIN {X 0,Y 239.952,Z 782.863,A -85,B 0,C 180,E1 -19175.232,E2 -19175.232} C_VEL
LIN {X 0,Y 240.2,Z 783.403,A -85,B 0,C 180,E1 -19176.723,E2 -19176.723} C_VEL
LIN {X 0,Y 240.571,Z 783.518,A -85,B 0,C 180,E1 -19178.401,E2 -19178.401} C_VEL
LIN {X 0,Y 241.223,Z 783.092,A -85,B 0,C 180,E1 -19180.069,E2 -19180.069} C_VEL
LIN {X 0,Y 242.058,Z 782.085,A -85,B 0,C 180,E1 -19181.728,E2 -19181.728} C_VEL
LIN {X 0,Y 243.616,Z 779.526,A -85,B 0,C 180,E1 -19184.196,E2 -19184.196} C_VEL
LIN {X 0,Y 245.578,Z 775.638,A -85,B 0,C 180,E1 -19186.631,E2 -19186.631} C_VEL
LIN {X 0,Y 248.211,Z 770.358,A -85,B 0,C 180,E1 -19189.004,E2 -19189.004} C_VEL
LIN {X 0,Y 250.623,Z 764.585,A -85,B 0,C 180,E1 -19190.95,E2 -19190.95} C_VEL
LIN {X 0,Y 253.333,Z 757.46,A -85,B 0,C 180,E1 -19192.856,E2 -19192.856} C_VEL
LIN {X 0,Y 256.207,Z 748.906,A -85,B 0,C 180,E1 -19194.671,E2 -19194.671} C_VEL
LIN {X 0,Y 259.165,Z 738.465,A -85,B 0,C 180,E1 -19196.364,E2 -19196.364} C_VEL
LIN {X 0,Y 261.909,Z 726.915,A -85,B 0,C 180,E1 -19197.792,E2 -19197.792} C_VEL
LIN {X 0,Y 263.982,Z 715.44,A -85,B 0,C 180,E1 -19198.853,E2 -19198.853} C_VEL
LIN {X 0,Y 266.071,Z 699.069,A -85,B 0,C 180,E1 -19199.942,E2 -19199.942} C_VEL
LIN {X 0,Y 270.968,Z 665.23,A -85,B 0,C 180,E1 -19201.739,E2 -19201.739} C_VEL
LIN {X 0,Y 275.674,Z 635.226,A -85,B 0,C 180,E1 -19203.239,E2 -19203.239} C_VEL
LIN {X 0,Y 276.254,Z 631.738,A -85,B 0,C 180,E1 -19203.488,E2 -19203.488} C_VEL
LIN {X 0,Y 278.523,Z 626.517,A -85,B 0,C 180,E1 -19204.036,E2 -19204.036} C_VEL
LIN {X 0,Y 280.255,Z 621.767,A -85,B 0,C 180,E1 -19204.743,E2 -19204.743} C_VEL
LIN {X 0,Y 280.341,Z 620.368,A -85,B 0,C 180,E1 -19205.213,E2 -19205.213} C_VEL
LIN {X 0,Y 280.072,Z 618.92,A -85,B 0,C 180,E1 -19205.949,E2 -19205.949} C_VEL
LIN {X 0,Y 278.354,Z 616.5,A -85,B 0,C 180,E1 -19208.491,E2 -19208.491} C_VEL
LIN {X 0,Y 276.968,Z 615.369,A -85,B 0,C 180,E1 -19211.282,E2 -19211.282} C_VEL
LIN {X 0,Y 276.307,Z 615.403,A -85,B 0,C 180,E1 -19213.375,E2 -19213.375} C_VEL
LIN {X 0,Y 275.849,Z 616.271,A -85,B 0,C 180,E1 -19215.512,E2 -19215.512} C_VEL
LIN {X 0,Y 275.493,Z 618.808,A -85,B 0,C 180,E1 -19218.45,E2 -19218.45} C_VEL
LIN {X 0,Y 275.289,Z 621.339,A -85,B 0,C 180,E1 -19220.339,E2 -19220.339} C_VEL
LIN {X 0,Y 274.945,Z 625.059,A -85,B 0,C 180,E1 -19222.412,E2 -19222.412} C_VEL
LIN {X 0,Y 274.775,Z 626.384,A -85,B 0,C 180,E1 -19223.029,E2 -19223.029} C_VEL
LIN {X 0,Y 272.341,Z 632.689,A -85,B 0,C 180,E1 -19224.732,E2 -19224.732} C_VEL
LIN {X 0,Y 273.237,Z 646.238,A -85,B 0,C 180,E1 -19226.977,E2 -19226.977} C_VEL
LIN {X 0,Y 274.181,Z 659.895,A -85,B 0,C 180,E1 -19228.864,E2 -19228.864} C_VEL
LIN {X 0,Y 274.654,Z 670.544,A -85,B 0,C 180,E1 -19230.067,E2 -19230.067} C_VEL
LIN {X 0,Y 274.534,Z 672.982,A -85,B 0,C 180,E1 -19230.261,E2 -19230.261} C_VEL
LIN {X 0,Y 269.334,Z 709.292,A -85,B 0,C 180,E1 -19232.039,E2 -19232.039} C_VEL
LIN {X 0,Y 267.212,Z 720.239,A -85,B 0,C 180,E1 -19232.807,E2 -19232.807} C_VEL
LIN {X 0,Y 264.664,Z 730.349,A -85,B 0,C 180,E1 -19233.802,E2 -19233.802} C_VEL
LIN {X 0,Y 261.52,Z 740.987,A -85,B 0,C 180,E1 -19235.172,E2 -19235.172} C_VEL
LIN {X 0,Y 258.872,Z 748.411,A -85,B 0,C 180,E1 -19236.394,E2 -19236.394} C_VEL
LIN {X 0,Y 256.1,Z 755.399,A -85,B 0,C 180,E1 -19237.831,E2 -19237.831} C_VEL
LIN {X 0,Y 253.002,Z 762.5,A -85,B 0,C 180,E1 -19239.682,E2 -19239.682} C_VEL
LIN {X 0,Y 250.71,Z 767.138,A -85,B 0,C 180,E1 -19241.194,E2 -19241.194} C_VEL
LIN {X 0,Y 247.61,Z 772.546,A -85,B 0,C 180,E1 -19243.511,E2 -19243.511} C_VEL
LIN {X 0,Y 245.13,Z 776.433,A -85,B 0,C 180,E1 -19245.895,E2 -19245.895} C_VEL
LIN {X 0,Y 243.192,Z 779.006,A -85,B 0,C 180,E1 -19248.329,E2 -19248.329} C_VEL
LIN {X 0,Y 242.111,Z 779.976,A -85,B 0,C 180,E1 -19249.97,E2 -19249.97} C_VEL
LIN {X 0,Y 240.937,Z 780.351,A -85,B 0,C 180,E1 -19252.648,E2 -19252.648} C_VEL
LIN {X 0,Y 240.207,Z 779.53,A -85,B 0,C 180,E1 -19254.964,E2 -19254.964} C_VEL
LIN {X 0,Y 240.001,Z 778.296,A -85,B 0,C 180,E1 -19256.643,E2 -19256.643} C_VEL
LIN {X 0,Y 239.873,Z 775.298,A -85,B 0,C 180,E1 -19259.161,E2 -19259.161} C_VEL
LIN {X 0,Y 239.948,Z 770.906,A -85,B 0,C 180,E1 -19261.679,E2 -19261.679} C_VEL
LIN {X 0,Y 240.242,Z 765.88,A -85,B 0,C 180,E1 -19263.774,E2 -19263.774} C_VEL
LIN {X 0,Y 240.358,Z 759.927,A -85,B 0,C 180,E1 -19265.712,E2 -19265.712} C_VEL
LIN {X 0,Y 240.792,Z 752.974,A -85,B 0,C 180,E1 -19267.547,E2 -19267.547} C_VEL
LIN {X 0,Y 241.284,Z 743.835,A -85,B 0,C 180,E1 -19269.43,E2 -19269.43} C_VEL
LIN {X 0,Y 241.696,Z 734.887,A -85,B 0,C 180,E1 -19270.895,E2 -19270.895} C_VEL
LIN {X 0,Y 242.246,Z 725.186,A -85,B 0,C 180,E1 -19272.142,E2 -19272.142} C_VEL
LIN {X 0,Y 242.594,Z 715.552,A -85,B 0,C 180,E1 -19273.081,E2 -19273.081} C_VEL
LIN {X 0,Y 243.049,Z 703.973,A -85,B 0,C 180,E1 -19273.908,E2 -19273.908} C_VEL
LIN {X 0,Y 244.121,Z 655.563,A -85,B 0,C 180,E1 -19276.275,E2 -19276.275} C_VEL
LIN {X 0,Y 242.735,Z 633.173,A -85,B 0,C 180,E1 -19277.355,E2 -19277.355} C_VEL
LIN {X 0,Y 242.779,Z 631.981,A -85,B 0,C 180,E1 -19277.46,E2 -19277.46} C_VEL
LIN {X 0,Y 244.156,Z 614.152,A -85,B 0,C 180,E1 -19281.531,E2 -19281.531} C_VEL
LIN {X 0,Y 245.836,Z 595.217,A -85,B 0,C 180,E1 -19285.847,E2 -19285.847} C_VEL
LIN {X 0,Y 247.31,Z 579.809,A -85,B 0,C 180,E1 -19289.354,E2 -19289.354} C_VEL
LIN {X 0,Y 244.34,Z 565.34,A -85,B 0,C 180,E1 -19292.882,E2 -19292.882} C_VEL
LIN {X 0,Y 242.095,Z 554.48,A -85,B 0,C 180,E1 -19295.675,E2 -19295.675} C_VEL
LIN {X 0,Y 241.961,Z 554.33,A -85,B 0,C 180,E1 -19299.718,E2 -19299.718} C_VEL
LIN {X 0,Y 241.94,Z 554.3,A -85,B 0,C 180,E1 -19304.2,E2 -19304.2} C_VEL
LIN {X 0,Y 241.961,Z 554.332,A -85,B 0,C 180,E1 -19308.081,E2 -19308.081} C_VEL
LIN {X 0,Y 241.994,Z 554.32,A -85,B 0,C 180,E1 -19312.417,E2 -19312.417} C_VEL
LIN {X 0,Y 242.031,Z 554.443,A -85,B 0,C 180,E1 -19314.866,E2 -19314.866} C_VEL
LIN {X 0,Y 242.499,Z 556.233,A -85,B 0,C 180,E1 -19315.638,E2 -19315.638} C_VEL
LIN {X 0,Y 250.254,Z 571.286,A -85,B 0,C 180,E1 -19317.406,E2 -19317.406} C_VEL
LIN {X 0,Y 257.286,Z 586.847,A -85,B 0,C 180,E1 -19318.91,E2 -19318.91} C_VEL
LIN {X 0,Y 261.173,Z 596.864,A -85,B 0,C 180,E1 -19319.741,E2 -19319.741} C_VEL
LIN {X 0,Y 258.946,Z 661.574,A -85,B 0,C 180,E1 -19321.505,E2 -19321.505} C_VEL
LIN {X 0,Y 257.894,Z 674.87,A -85,B 0,C 180,E1 -19322.132,E2 -19322.132} C_VEL
LIN {X 0,Y 256.465,Z 688.259,A -85,B 0,C 180,E1 -19323.117,E2 -19323.117} C_VEL
LIN {X 0,Y 254.813,Z 699.56,A -85,B 0,C 180,E1 -19324.251,E2 -19324.251} C_VEL
LIN {X 0,Y 252.672,Z 711.197,A -85,B 0,C 180,E1 -19325.777,E2 -19325.777} C_VEL
LIN {X 0,Y 250.445,Z 721.965,A -85,B 0,C 180,E1 -19327.585,E2 -19327.585} C_VEL
LIN {X 0,Y 248.333,Z 731.863,A -85,B 0,C 180,E1 -19329.714,E2 -19329.714} C_VEL
LIN {X 0,Y 246.018,Z 740.771,A -85,B 0,C 180,E1 -19332.114,E2 -19332.114} C_VEL
LIN {X 0,Y 244.156,Z 747.937,A -85,B 0,C 180,E1 -19334.557,E2 -19334.557} C_VEL
LIN {X 0,Y 242.864,Z 752.77,A -85,B 0,C 180,E1 -19336.613,E2 -19336.613} C_VEL
LIN {X 0,Y 241.618,Z 757.464,A -85,B 0,C 180,E1 -19339.1,E2 -19339.1} C_VEL
LIN {X 0,Y 240.808,Z 761.049,A -85,B 0,C 180,E1 -19341.608,E2 -19341.608} C_VEL
LIN {X 0,Y 240.32,Z 763.43,A -85,B 0,C 180,E1 -19343.888,E2 -19343.888} C_VEL
LIN {X 0,Y 240.036,Z 765.283,A -85,B 0,C 180,E1 -19346.641,E2 -19346.641} C_VEL
LIN {X 0,Y 239.924,Z 766.122,A -85,B 0,C 180,E1 -19349.998,E2 -19349.998} C_VEL
LIN {X 0,Y 239.919,Z 765.93,A -85,B 0,C 180,E1 -19351.677,E2 -19351.677} C_VEL
LIN {X 0,Y 240.033,Z 765.345,A -85,B 0,C 180,E1 -19353.356,E2 -19353.356} C_VEL
LIN {X 0,Y 240.449,Z 763.025,A -85,B 0,C 180,E1 -19356.713,E2 -19356.713} C_VEL
LIN {X 0,Y 241.037,Z 760.157,A -85,B 0,C 180,E1 -19359.227,E2 -19359.227} C_VEL
LIN {X 0,Y 241.963,Z 756.266,A -85,B 0,C 180,E1 -19361.73,E2 -19361.73} C_VEL
LIN {X 0,Y 243.288,Z 751.247,A -85,B 0,C 180,E1 -19364.212,E2 -19364.212} C_VEL
LIN {X 0,Y 244.885,Z 744.927,A -85,B 0,C 180,E1 -19366.676,E2 -19366.676} C_VEL
LIN {X 0,Y 247.048,Z 737.009,A -85,B 0,C 180,E1 -19369.094,E2 -19369.094} C_VEL
LIN {X 0,Y 249.189,Z 728.145,A -85,B 0,C 180,E1 -19371.268,E2 -19371.268} C_VEL
LIN {X 0,Y 251.311,Z 717.997,A -85,B 0,C 180,E1 -19373.265,E2 -19373.265} C_VEL
LIN {X 0,Y 253.585,Z 706.587,A -85,B 0,C 180,E1 -19375,E2 -19375} C_VEL
LIN {X 0,Y 255.513,Z 695.369,A -85,B 0,C 180,E1 -19376.327,E2 -19376.327} C_VEL
LIN {X 0,Y 257.217,Z 682.701,A -85,B 0,C 180,E1 -19377.455,E2 -19377.455} C_VEL
LIN {X 0,Y 258.461,Z 670.001,A -85,B 0,C 180,E1 -19378.247,E2 -19378.247} C_VEL
LIN {X 0,Y 259.246,Z 656.885,A -85,B 0,C 180,E1 -19378.761,E2 -19378.761} C_VEL
LIN {X 0,Y 261.244,Z 596.973,A -85,B 0,C 180,E1 -19380.377,E2 -19380.377} C_VEL
LIN {X 0,Y 254.717,Z 580.891,A -85,B 0,C 180,E1 -19381.77,E2 -19381.77} C_VEL
LIN {X 0,Y 247.507,Z 565.945,A -85,B 0,C 180,E1 -19383.325,E2 -19383.325} C_VEL
LIN {X 0,Y 242.475,Z 556.117,A -85,B 0,C 180,E1 -19384.519,E2 -19384.519} C_VEL
LIN {X 0,Y 242.038,Z 554.426,A -85,B 0,C 180,E1 -19385.319,E2 -19385.319} C_VEL
LIN {X 0,Y 241.969,Z 554.329,A -85,B 0,C 180,E1 -19389.714,E2 -19389.714} C_VEL
LIN {X 0,Y 241.928,Z 554.329,A -85,B 0,C 180,E1 -19394.2,E2 -19394.2} C_VEL
LIN {X 0,Y 241.95,Z 554.347,A -85,B 0,C 180,E1 -19398.08,E2 -19398.08} C_VEL
LIN {X 0,Y 242.007,Z 554.311,A -85,B 0,C 180,E1 -19402.421,E2 -19402.421} C_VEL
LIN {X 0,Y 241.986,Z 554.339,A -85,B 0,C 180,E1 -19406.508,E2 -19406.508} C_VEL
LIN {X 0,Y 242.031,Z 554.336,A -85,B 0,C 180,E1 -19410.586,E2 -19410.586} C_VEL
LIN {X 0,Y 242.062,Z 554.332,A -85,B 0,C 180,E1 -19414.182,E2 -19414.182} C_VEL
LIN {X 0,Y 242.047,Z 554.32,A -85,B 0,C 180,E1 -19418.296,E2 -19418.296} C_VEL
LIN {X 0,Y 242.157,Z 554.305,A -85,B 0,C 180,E1 -19423.278,E2 -19423.278} C_VEL
LIN {X 0,Y 242.18,Z 554.312,A -85,B 0,C 180,E1 -19428.279,E2 -19428.279} C_VEL
LIN {X 0,Y 242.421,Z 554.277,A -85,B 0,C 180,E1 -19431.665,E2 -19431.665} C_VEL
LIN {X 0,Y 242.255,Z 554.303,A -85,B 0,C 180,E1 -19435.007,E2 -19435.007} C_VEL
LIN {X 0,Y 242.388,Z 554.273,A -85,B 0,C 180,E1 -19436.865,E2 -19436.865} C_VEL
LIN {X 0,Y 241.827,Z 554.352,A -85,B 0,C 180,E1 -19438.256,E2 -19438.256} C_VEL
LIN {X 0,Y 240.273,Z 554.555,A -85,B 0,C 180,E1 -19439.622,E2 -19439.622} C_VEL
LIN {X 0,Y 236.463,Z 555.019,A -85,B 0,C 180,E1 -19442.37,E2 -19442.37} C_VEL
LIN {X 0,Y 235.344,Z 555.151,A -85,B 0,C 180,E1 -19443.805,E2 -19443.805} C_VEL
LIN {X 0,Y 235.236,Z 555.166,A -85,B 0,C 180,E1 -19444.293,E2 -19444.293} C_VEL
LIN {X 0,Y 235.399,Z 555.162,A -85,B 0,C 180,E1 -19446.859,E2 -19446.859} C_VEL
LIN {X 0,Y 235.247,Z 555.164,A -85,B 0,C 180,E1 -19450.326,E2 -19450.326} C_VEL
LIN {X 0,Y 235.107,Z 555.184,A -85,B 0,C 180,E1 -19455.607,E2 -19455.607} C_VEL
LIN {X 0,Y 235.003,Z 555.213,A -85,B 0,C 180,E1 -19459.206,E2 -19459.206} C_VEL
LIN {X 0,Y 234.955,Z 555.212,A -85,B 0,C 180,E1 -19462.883,E2 -19462.883} C_VEL
LIN {X 0,Y 234.961,Z 555.205,A -85,B 0,C 180,E1 -19466.658,E2 -19466.658} C_VEL
LIN {X 0,Y 234.916,Z 555.216,A -85,B 0,C 180,E1 -19470.57,E2 -19470.57} C_VEL
LIN {X 0,Y 234.921,Z 555.208,A -85,B 0,C 180,E1 -19474.64,E2 -19474.64} C_VEL
LIN {X 0,Y 234.936,Z 555.215,A -85,B 0,C 180,E1 -19478.946,E2 -19478.946} C_VEL
LIN {X 0,Y 234.922,Z 555.206,A -85,B 0,C 180,E1 -19483.478,E2 -19483.478} C_VEL
LIN {X 0,Y 234.97,Z 555.203,A -85,B 0,C 180,E1 -19486.536,E2 -19486.536} C_VEL
LIN {X 0,Y 234.97,Z 555.249,A -85,B 0,C 180,E1 -19489.065,E2 -19489.065} C_VEL
LIN {X 0,Y 236.1,Z 559.501,A -85,B 0,C 180,E1 -19491.312,E2 -19491.312} C_VEL
LIN {X 0,Y 237.92,Z 567.072,A -85,B 0,C 180,E1 -19494.754,E2 -19494.754} C_VEL
LIN {X 0,Y 245.33,Z 582.748,A -85,B 0,C 180,E1 -19496.555,E2 -19496.555} C_VEL
LIN {X 0,Y 251.265,Z 597.04,A -85,B 0,C 180,E1 -19497.911,E2 -19497.911} C_VEL
LIN {X 0,Y 254.495,Z 619.576,A -85,B 0,C 180,E1 -19499.09,E2 -19499.09} C_VEL
LIN {X 0,Y 252.335,Z 675.78,A -85,B 0,C 180,E1 -19500.66,E2 -19500.66} C_VEL
LIN {X 0,Y 251.088,Z 689.663,A -85,B 0,C 180,E1 -19501.36,E2 -19501.36} C_VEL
LIN {X 0,Y 249.39,Z 702.096,A -85,B 0,C 180,E1 -19502.293,E2 -19502.293} C_VEL
LIN {X 0,Y 247.265,Z 714.787,A -85,B 0,C 180,E1 -19503.636,E2 -19503.636} C_VEL
LIN {X 0,Y 244.922,Z 726.059,A -85,B 0,C 180,E1 -19505.189,E2 -19505.189} C_VEL
LIN {X 0,Y 242.591,Z 736.217,A -85,B 0,C 180,E1 -19506.979,E2 -19506.979} C_VEL
LIN {X 0,Y 240.391,Z 745.376,A -85,B 0,C 180,E1 -19509.016,E2 -19509.016} C_VEL
LIN {X 0,Y 238.156,Z 754.304,A -85,B 0,C 180,E1 -19511.506,E2 -19511.506} C_VEL
LIN {X 0,Y 236.223,Z 761.489,A -85,B 0,C 180,E1 -19514.028,E2 -19514.028} C_VEL
LIN {X 0,Y 234.525,Z 768.033,A -85,B 0,C 180,E1 -19517.013,E2 -19517.013} C_VEL
LIN {X 0,Y 233.59,Z 772.371,A -85,B 0,C 180,E1 -19519.602,E2 -19519.602} C_VEL
LIN {X 0,Y 233.181,Z 774.673,A -85,B 0,C 180,E1 -19521.334,E2 -19521.334} C_VEL
LIN {X 0,Y 232.889,Z 776.536,A -85,B 0,C 180,E1 -19523.069,E2 -19523.069} C_VEL
LIN {X 0,Y 232.684,Z 778.303,A -85,B 0,C 180,E1 -19525.37,E2 -19525.37} C_VEL
LIN {X 0,Y 232.745,Z 779.54,A -85,B 0,C 180,E1 -19528.271,E2 -19528.271} C_VEL
LIN {X 0,Y 232.782,Z 779.753,A -85,B 0,C 180,E1 -19530.002,E2 -19530.002} C_VEL
LIN {X 0,Y 232.819,Z 779.556,A -85,B 0,C 180,E1 -19532.164,E2 -19532.164} C_VEL
LIN {X 0,Y 232.882,Z 782.339,A -85,B 0,C 180,E1 -19535.196,E2 -19535.196} C_VEL
LIN {X 0,Y 233.132,Z 783.212,A -85,B 0,C 180,E1 -19536.927,E2 -19536.927} C_VEL
LIN {X 0,Y 233.538,Z 783.502,A -85,B 0,C 180,E1 -19538.656,E2 -19538.656} C_VEL
LIN {X 0,Y 234.234,Z 783.216,A -85,B 0,C 180,E1 -19540.373,E2 -19540.373} C_VEL
LIN {X 0,Y 235.112,Z 782.407,A -85,B 0,C 180,E1 -19542.08,E2 -19542.08} C_VEL
LIN {X 0,Y 236.175,Z 781.082,A -85,B 0,C 180,E1 -19543.774,E2 -19543.774} C_VEL
LIN {X 0,Y 238.127,Z 778.078,A -85,B 0,C 180,E1 -19546.284,E2 -19546.284} C_VEL
LIN {X 0,Y 239.799,Z 775.286,A -85,B 0,C 180,E1 -19547.924,E2 -19547.924} C_VEL
LIN {X 0,Y 242.703,Z 769.966,A -85,B 0,C 180,E1 -19550.335,E2 -19550.335} C_VEL
LIN {X 0,Y 245.415,Z 764.171,A -85,B 0,C 180,E1 -19552.301,E2 -19552.301} C_VEL
LIN {X 0,Y 248.326,Z 756.999,A -85,B 0,C 180,E1 -19554.23,E2 -19554.23} C_VEL
LIN {X 0,Y 251.581,Z 748.446,A -85,B 0,C 180,E1 -19556.044,E2 -19556.044} C_VEL
LIN {X 0,Y 254.437,Z 739.225,A -85,B 0,C 180,E1 -19557.561,E2 -19557.561} C_VEL
LIN {X 0,Y 257.457,Z 728.124,A -85,B 0,C 180,E1 -19558.983,E2 -19558.983} C_VEL
LIN {X 0,Y 259.687,Z 717.564,A -85,B 0,C 180,E1 -19560,E2 -19560} C_VEL
LIN {X 0,Y 261.273,Z 707.695,A -85,B 0,C 180,E1 -19560.737,E2 -19560.737} C_VEL
LIN {X 0,Y 265.766,Z 677.193,A -85,B 0,C 180,E1 -19562.491,E2 -19562.491} C_VEL
LIN {X 0,Y 272.508,Z 637.103,A -85,B 0,C 180,E1 -19564.513,E2 -19564.513} C_VEL
LIN {X 0,Y 273.374,Z 631.897,A -85,B 0,C 180,E1 -19564.882,E2 -19564.882} C_VEL
LIN {X 0,Y 275.455,Z 627.058,A -85,B 0,C 180,E1 -19565.453,E2 -19565.453} C_VEL
LIN {X 0,Y 276.006,Z 625.229,A -85,B 0,C 180,E1 -19565.85,E2 -19565.85} C_VEL
LIN {X 0,Y 275.59,Z 624.036,A -85,B 0,C 180,E1 -19566.628,E2 -19566.628} C_VEL
LIN {X 0,Y 274.692,Z 622.859,A -85,B 0,C 180,E1 -19567.883,E2 -19567.883} C_VEL
LIN {X 0,Y 273.489,Z 621.581,A -85,B 0,C 180,E1 -19569.975,E2 -19569.975} C_VEL
LIN {X 0,Y 272.537,Z 621.098,A -85,B 0,C 180,E1 -19572.105,E2 -19572.105} C_VEL
LIN {X 0,Y 271.893,Z 621.387,A -85,B 0,C 180,E1 -19574.261,E2 -19574.261} C_VEL
LIN {X 0,Y 271.361,Z 622.679,A -85,B 0,C 180,E1 -19576.485,E2 -19576.485} C_VEL
LIN {X 0,Y 270.95,Z 624.955,A -85,B 0,C 180,E1 -19578.784,E2 -19578.784} C_VEL
LIN {X 0,Y 270.676,Z 627.096,A -85,B 0,C 180,E1 -19580.341,E2 -19580.341} C_VEL
LIN {X 0,Y 270.139,Z 630.61,A -85,B 0,C 180,E1 -19582.285,E2 -19582.285} C_VEL
LIN {X 0,Y 269.286,Z 633.146,A -85,B 0,C 180,E1 -19582.991,E2 -19582.991} C_VEL
LIN {X 0,Y 269.732,Z 645.912,A -85,B 0,C 180,E1 -19585.26,E2 -19585.26} C_VEL
LIN {X 0,Y 270.247,Z 657.549,A -85,B 0,C 180,E1 -19587.031,E2 -19587.031} C_VEL
LIN {X 0,Y 270.681,Z 670.469,A -85,B 0,C 180,E1 -19588.678,E2 -19588.678} C_VEL
LIN {X 0,Y 270.605,Z 674.171,A -85,B 0,C 180,E1 -19589.045,E2 -19589.045} C_VEL
LIN {X 0,Y 265.288,Z 708.905,A -85,B 0,C 180,E1 -19590.762,E2 -19590.762} C_VEL
LIN {X 0,Y 262.927,Z 720.281,A -85,B 0,C 180,E1 -19591.567,E2 -19591.567} C_VEL
LIN {X 0,Y 259.988,Z 731.144,A -85,B 0,C 180,E1 -19592.642,E2 -19592.642} C_VEL
LIN {X 0,Y 256.645,Z 741.576,A -85,B 0,C 180,E1 -19594.014,E2 -19594.014} C_VEL
LIN {X 0,Y 253.456,Z 749.746,A -85,B 0,C 180,E1 -19595.422,E2 -19595.422} C_VEL
LIN {X 0,Y 250.497,Z 756.507,A -85,B 0,C 180,E1 -19596.872,E2 -19596.872} C_VEL
LIN {X 0,Y 247.196,Z 763.429,A -85,B 0,C 180,E1 -19598.747,E2 -19598.747} C_VEL
LIN {X 0,Y 244.154,Z 768.813,A -85,B 0,C 180,E1 -19600.669,E2 -19600.669} C_VEL
LIN {X 0,Y 240.912,Z 773.8,A -85,B 0,C 180,E1 -19603.039,E2 -19603.039} C_VEL
LIN {X 0,Y 239.058,Z 776.293,A -85,B 0,C 180,E1 -19604.658,E2 -19604.658} C_VEL
LIN {X 0,Y 237.548,Z 778.159,A -85,B 0,C 180,E1 -19606.309,E2 -19606.309} C_VEL
LIN {X 0,Y 236.268,Z 779.469,A -85,B 0,C 180,E1 -19607.982,E2 -19607.982} C_VEL
LIN {X 0,Y 235.152,Z 780.251,A -85,B 0,C 180,E1 -19609.67,E2 -19609.67} C_VEL
LIN {X 0,Y 234.327,Z 780.495,A -85,B 0,C 180,E1 -19611.375,E2 -19611.375} C_VEL
LIN {X 0,Y 233.666,Z 780.149,A -85,B 0,C 180,E1 -19613.09,E2 -19613.09} C_VEL
LIN {X 0,Y 233.147,Z 779.228,A -85,B 0,C 180,E1 -19614.812,E2 -19614.812} C_VEL
LIN {X 0,Y 232.878,Z 776.9,A -85,B 0,C 180,E1 -19617.406,E2 -19617.406} C_VEL
LIN {X 0,Y 232.849,Z 773.071,A -85,B 0,C 180,E1 -19620,E2 -19620} C_VEL
LIN {X 0,Y 233.063,Z 767.762,A -85,B 0,C 180,E1 -19622.593,E2 -19622.593} C_VEL
LIN {X 0,Y 233.257,Z 761.831,A -85,B 0,C 180,E1 -19624.753,E2 -19624.753} C_VEL
LIN {X 0,Y 233.574,Z 755.645,A -85,B 0,C 180,E1 -19626.55,E2 -19626.55} C_VEL
LIN {X 0,Y 233.941,Z 748.43,A -85,B 0,C 180,E1 -19628.268,E2 -19628.268} C_VEL
LIN {X 0,Y 234.338,Z 739.816,A -85,B 0,C 180,E1 -19629.93,E2 -19629.93} C_VEL
LIN {X 0,Y 234.948,Z 729.675,A -85,B 0,C 180,E1 -19631.43,E2 -19631.43} C_VEL
LIN {X 0,Y 235.465,Z 718.307,A -85,B 0,C 180,E1 -19632.716,E2 -19632.716} C_VEL
LIN {X 0,Y 235.818,Z 707.565,A -85,B 0,C 180,E1 -19633.574,E2 -19633.574} C_VEL
LIN {X 0,Y 236.279,Z 689.79,A -85,B 0,C 180,E1 -19634.535,E2 -19634.535} C_VEL
LIN {X 0,Y 236.995,Z 655.352,A -85,B 0,C 180,E1 -19636.28,E2 -19636.28} C_VEL
LIN {X 0,Y 235.641,Z 633.342,A -85,B 0,C 180,E1 -19637.393,E2 -19637.393} C_VEL
LIN {X 0,Y 235.69,Z 631.971,A -85,B 0,C 180,E1 -19637.53,E2 -19637.53} C_VEL
LIN {X 0,Y 237.106,Z 613.896,A -85,B 0,C 180,E1 -19641.747,E2 -19641.747} C_VEL
LIN {X 0,Y 238.843,Z 594.829,A -85,B 0,C 180,E1 -19646.192,E2 -19646.192} C_VEL
LIN {X 0,Y 240.243,Z 581.068,A -85,B 0,C 180,E1 -19649.39,E2 -19649.39} C_VEL
LIN {X 0,Y 238.417,Z 571.594,A -85,B 0,C 180,E1 -19651.738,E2 -19651.738} C_VEL
LIN {X 0,Y 235.085,Z 555.384,A -85,B 0,C 180,E1 -19655.918,E2 -19655.918} C_VEL
LIN {X 0,Y 234.947,Z 555.216,A -85,B 0,C 180,E1 -19658.944,E2 -19658.944} C_VEL
LIN {X 0,Y 234.895,Z 555.169,A -85,B 0,C 180,E1 -19663.485,E2 -19663.485} C_VEL
LIN {X 0,Y 234.955,Z 555.216,A -85,B 0,C 180,E1 -19666.528,E2 -19666.528} C_VEL
LIN {X 0,Y 234.928,Z 555.183,A -85,B 0,C 180,E1 -19671.079,E2 -19671.079} C_VEL
LIN {X 0,Y 234.983,Z 555.43,A -85,B 0,C 180,E1 -19674.023,E2 -19674.023} C_VEL
LIN {X 0,Y 235.313,Z 556.708,A -85,B 0,C 180,E1 -19674.458,E2 -19674.458} C_VEL
LIN {X 0,Y 241.782,Z 568.663,A -85,B 0,C 180,E1 -19676.009,E2 -19676.009} C_VEL
LIN {X 0,Y 249.211,Z 584.266,A -85,B 0,C 180,E1 -19677.687,E2 -19677.687} C_VEL
LIN {X 0,Y 255.021,Z 598.552,A -85,B 0,C 180,E1 -19678.978,E2 -19678.978} C_VEL
LIN {X 0,Y 252.719,Z 662.491,A -85,B 0,C 180,E1 -19680.767,E2 -19680.767} C_VEL
LIN {X 0,Y 251.588,Z 675.91,A -85,B 0,C 180,E1 -19681.432,E2 -19681.432} C_VEL
LIN {X 0,Y 250.161,Z 688.471,A -85,B 0,C 180,E1 -19682.382,E2 -19682.382} C_VEL
LIN {X 0,Y 248.45,Z 699.77,A -85,B 0,C 180,E1 -19683.542,E2 -19683.542} C_VEL
LIN {X 0,Y 246.22,Z 711.405,A -85,B 0,C 180,E1 -19685.1,E2 -19685.1} C_VEL
LIN {X 0,Y 243.901,Z 722.173,A -85,B 0,C 180,E1 -19686.949,E2 -19686.949} C_VEL
LIN {X 0,Y 242.002,Z 730.679,A -85,B 0,C 180,E1 -19688.788,E2 -19688.788} C_VEL
LIN {X 0,Y 239.635,Z 739.631,A -85,B 0,C 180,E1 -19691.178,E2 -19691.178} C_VEL
LIN {X 0,Y 237.564,Z 747.036,A -85,B 0,C 180,E1 -19693.676,E2 -19693.676} C_VEL
LIN {X 0,Y 235.946,Z 752.977,A -85,B 0,C 180,E1 -19696.213,E2 -19696.213} C_VEL
LIN {X 0,Y 234.646,Z 757.67,A -85,B 0,C 180,E1 -19698.772,E2 -19698.772} C_VEL
LIN {X 0,Y 233.795,Z 761.254,A -85,B 0,C 180,E1 -19701.354,E2 -19701.354} C_VEL
LIN {X 0,Y 233.226,Z 763.837,A -85,B 0,C 180,E1 -19703.945,E2 -19703.945} C_VEL
LIN {X 0,Y 232.96,Z 765.487,A -85,B 0,C 180,E1 -19706.539,E2 -19706.539} C_VEL
LIN {X 0,Y 232.835,Z 766.326,A -85,B 0,C 180,E1 -19709.998,E2 -19709.998} C_VEL
LIN {X 0,Y 232.835,Z 766.134,A -85,B 0,C 180,E1 -19711.728,E2 -19711.728} C_VEL
LIN {X 0,Y 232.958,Z 765.549,A -85,B 0,C 180,E1 -19713.458,E2 -19713.458} C_VEL
LIN {X 0,Y 233.387,Z 763.229,A -85,B 0,C 180,E1 -19716.917,E2 -19716.917} C_VEL
LIN {X 0,Y 234.03,Z 760.361,A -85,B 0,C 180,E1 -19719.505,E2 -19719.505} C_VEL
LIN {X 0,Y 235.014,Z 756.469,A -85,B 0,C 180,E1 -19722.082,E2 -19722.082} C_VEL
LIN {X 0,Y 236.406,Z 751.451,A -85,B 0,C 180,E1 -19724.635,E2 -19724.635} C_VEL
LIN {X 0,Y 238.088,Z 745.13,A -85,B 0,C 180,E1 -19727.167,E2 -19727.167} C_VEL
LIN {X 0,Y 240.36,Z 737.211,A -85,B 0,C 180,E1 -19729.647,E2 -19729.647} C_VEL
LIN {X 0,Y 242.444,Z 728.895,A -85,B 0,C 180,E1 -19731.752,E2 -19731.752} C_VEL
LIN {X 0,Y 244.587,Z 719.296,A -85,B 0,C 180,E1 -19733.719,E2 -19733.719} C_VEL
LIN {X 0,Y 246.897,Z 708.209,A -85,B 0,C 180,E1 -19735.5,E2 -19735.5} C_VEL
LIN {X 0,Y 248.889,Z 697.33,A -85,B 0,C 180,E1 -19736.857,E2 -19736.857} C_VEL
LIN {X 0,Y 250.664,Z 685.298,A -85,B 0,C 180,E1 -19738.008,E2 -19738.008} C_VEL
LIN {X 0,Y 252.019,Z 672.926,A -85,B 0,C 180,E1 -19738.866,E2 -19738.866} C_VEL
LIN {X 0,Y 252.979,Z 660.073,A -85,B 0,C 180,E1 -19739.429,E2 -19739.429} C_VEL
LIN {X 0,Y 255.108,Z 598.697,A -85,B 0,C 180,E1 -19741.139,E2 -19741.139} C_VEL
LIN {X 0,Y 248.456,Z 582.517,A -85,B 0,C 180,E1 -19742.62,E2 -19742.62} C_VEL
LIN {X 0,Y 240.784,Z 566.785,A -85,B 0,C 180,E1 -19744.361,E2 -19744.361} C_VEL
LIN {X 0,Y 235.213,Z 556.368,A -85,B 0,C 180,E1 -19745.743,E2 -19745.743} C_VEL
LIN {X 0,Y 234.974,Z 555.281,A -85,B 0,C 180,E1 -19746.267,E2 -19746.267} C_VEL
LIN {X 0,Y 234.938,Z 555.208,A -85,B 0,C 180,E1 -19748.943,E2 -19748.943} C_VEL
LIN {X 0,Y 234.884,Z 555.213,A -85,B 0,C 180,E1 -19753.484,E2 -19753.484} C_VEL
LIN {X 0,Y 234.915,Z 555.211,A -85,B 0,C 180,E1 -19756.52,E2 -19756.52} C_VEL
LIN {X 0,Y 234.95,Z 555.185,A -85,B 0,C 180,E1 -19761.085,E2 -19761.085} C_VEL
LIN {X 0,Y 234.955,Z 555.221,A -85,B 0,C 180,E1 -19765.366,E2 -19765.366} C_VEL
LIN {X 0,Y 234.964,Z 555.217,A -85,B 0,C 180,E1 -19770.156,E2 -19770.156} C_VEL
LIN {X 0,Y 234.988,Z 555.208,A -85,B 0,C 180,E1 -19773.793,E2 -19773.793} C_VEL
LIN {X 0,Y 235.005,Z 555.201,A -85,B 0,C 180,E1 -19778.969,E2 -19778.969} C_VEL
LIN {X 0,Y 235.09,Z 555.186,A -85,B 0,C 180,E1 -19783.059,E2 -19783.059} C_VEL
LIN {X 0,Y 235.14,Z 555.19,A -85,B 0,C 180,E1 -19787.923,E2 -19787.923} C_VEL
LIN {X 0,Y 235.37,Z 555.153,A -85,B 0,C 180,E1 -19791.414,E2 -19791.414} C_VEL
LIN {X 0,Y 235.398,Z 555.162,A -85,B 0,C 180,E1 -19793.141,E2 -19793.141} C_VEL
LIN {X 0,Y 235.59,Z 555.128,A -85,B 0,C 180,E1 -19798.29,E2 -19798.29} C_VEL
LIN {X 0,Y 235.59,Z 555.132,A -85,B 0,C 180,E1 -19801.709,E2 -19801.709} C_VEL
LIN {X 0,Y 235.236,Z 555.166,A -85,B 0,C 180,E1 -19804.293,E2 -19804.293} C_VEL
LIN {X 0,Y 234.52,Z 555.268,A -85,B 0,C 180,E1 -19805.724,E2 -19805.724} C_VEL
LIN {X 0,Y 231.64,Z 555.626,A -85,B 0,C 180,E1 -19808.058,E2 -19808.058} C_VEL
LIN {X 0,Y 229.217,Z 555.918,A -85,B 0,C 180,E1 -19809.962,E2 -19809.962} C_VEL
LIN {X 0,Y 228.175,Z 556.051,A -85,B 0,C 180,E1 -19811.439,E2 -19811.439} C_VEL
LIN {X 0,Y 228.087,Z 556.064,A -85,B 0,C 180,E1 -19811.94,E2 -19811.94} C_VEL
LIN {X 0,Y 228.051,Z 556.062,A -85,B 0,C 180,E1 -19816.103,E2 -19816.103} C_VEL
LIN {X 0,Y 227.937,Z 556.09,A -85,B 0,C 180,E1 -19819.826,E2 -19819.826} C_VEL
LIN {X 0,Y 227.908,Z 556.094,A -85,B 0,C 180,E1 -19823.633,E2 -19823.633} C_VEL
LIN {X 0,Y 227.873,Z 556.092,A -85,B 0,C 180,E1 -19827.557,E2 -19827.557} C_VEL
LIN {X 0,Y 227.861,Z 556.094,A -85,B 0,C 180,E1 -19831.624,E2 -19831.624} C_VEL
LIN {X 0,Y 227.875,Z 556.071,A -85,B 0,C 180,E1 -19835.873,E2 -19835.873} C_VEL
LIN {X 0,Y 227.859,Z 556.1,A -85,B 0,C 180,E1 -19840.37,E2 -19840.37} C_VEL
LIN {X 0,Y 227.849,Z 556.105,A -85,B 0,C 180,E1 -19844.814,E2 -19844.814} C_VEL
LIN {X 0,Y 227.935,Z 556.216,A -85,B 0,C 180,E1 -19848.167,E2 -19848.167} C_VEL
LIN {X 0,Y 229.666,Z 562.782,A -85,B 0,C 180,E1 -19851.616,E2 -19851.616} C_VEL
LIN {X 0,Y 230.678,Z 566.88,A -85,B 0,C 180,E1 -19853.48,E2 -19853.48} C_VEL
LIN {X 0,Y 237.19,Z 580.338,A -85,B 0,C 180,E1 -19855.169,E2 -19855.169} C_VEL
LIN {X 0,Y 243.427,Z 594.386,A -85,B 0,C 180,E1 -19856.664,E2 -19856.664} C_VEL
LIN {X 0,Y 245.573,Z 600.061,A -85,B 0,C 180,E1 -19857.183,E2 -19857.183} C_VEL
LIN {X 0,Y 248.382,Z 620.802,A -85,B 0,C 180,E1 -19858.289,E2 -19858.289} C_VEL
LIN {X 0,Y 246.173,Z 675.591,A -85,B 0,C 180,E1 -19859.851,E2 -19859.851} C_VEL
LIN {X 0,Y 244.887,Z 689.468,A -85,B 0,C 180,E1 -19860.565,E2 -19860.565} C_VEL
LIN {X 0,Y 243.132,Z 701.898,A -85,B 0,C 180,E1 -19861.515,E2 -19861.515} C_VEL
LIN {X 0,Y 240.931,Z 714.587,A -85,B 0,C 180,E1 -19862.886,E2 -19862.886} C_VEL
LIN {X 0,Y 238.501,Z 725.858,A -85,B 0,C 180,E1 -19864.473,E2 -19864.473} C_VEL
LIN {X 0,Y 236.056,Z 736.015,A -85,B 0,C 180,E1 -19866.303,E2 -19866.303} C_VEL
LIN {X 0,Y 233.738,Z 745.172,A -85,B 0,C 180,E1 -19868.389,E2 -19868.389} C_VEL
LIN {X 0,Y 231.429,Z 754.102,A -85,B 0,C 180,E1 -19870.948,E2 -19870.948} C_VEL
LIN {X 0,Y 229.393,Z 761.285,A -85,B 0,C 180,E1 -19873.539,E2 -19873.539} C_VEL
LIN {X 0,Y 227.561,Z 767.828,A -85,B 0,C 180,E1 -19876.609,E2 -19876.609} C_VEL
LIN {X 0,Y 226.585,Z 772.167,A -85,B 0,C 180,E1 -19879.276,E2 -19879.276} C_VEL
LIN {X 0,Y 226.139,Z 774.468,A -85,B 0,C 180,E1 -19881.062,E2 -19881.062} C_VEL
LIN {X 0,Y 225.821,Z 776.331,A -85,B 0,C 180,E1 -19882.85,E2 -19882.85} C_VEL
LIN {X 0,Y 225.58,Z 778.299,A -85,B 0,C 180,E1 -19885.54,E2 -19885.54} C_VEL
LIN {X 0,Y 225.639,Z 779.335,A -85,B 0,C 180,E1 -19888.217,E2 -19888.217} C_VEL
LIN {X 0,Y 225.696,Z 779.549,A -85,B 0,C 180,E1 -19890.002,E2 -19890.002} C_VEL
LIN {X 0,Y 225.792,Z 779.23,A -85,B 0,C 180,E1 -19892.678,E2 -19892.678} C_VEL
LIN {X 0,Y 225.844,Z 781.831,A -85,B 0,C 180,E1 -19895.358,E2 -19895.358} C_VEL
LIN {X 0,Y 226.087,Z 782.836,A -85,B 0,C 180,E1 -19897.144,E2 -19897.144} C_VEL
LIN {X 0,Y 226.526,Z 783.316,A -85,B 0,C 180,E1 -19898.926,E2 -19898.926} C_VEL
LIN {X 0,Y 227.239,Z 783.284,A -85,B 0,C 180,E1 -19900.696,E2 -19900.696} C_VEL
LIN {X 0,Y 228.183,Z 782.75,A -85,B 0,C 180,E1 -19902.452,E2 -19902.452} C_VEL
LIN {X 0,Y 229.317,Z 781.692,A -85,B 0,C 180,E1 -19904.194,E2 -19904.194} C_VEL
LIN {X 0,Y 231.375,Z 778.984,A -85,B 0,C 180,E1 -19906.773,E2 -19906.773} C_VEL
LIN {X 0,Y 234.2,Z 775.022,A -85,B 0,C 180,E1 -19909.276,E2 -19909.276} C_VEL
LIN {X 0,Y 237.335,Z 769.671,A -85,B 0,C 180,E1 -19911.726,E2 -19911.726} C_VEL
LIN {X 0,Y 240.345,Z 763.878,A -85,B 0,C 180,E1 -19913.709,E2 -19913.709} C_VEL
LIN {X 0,Y 243.588,Z 756.754,A -85,B 0,C 180,E1 -19915.646,E2 -19915.646} C_VEL
LIN {X 0,Y 247.032,Z 748.408,A -85,B 0,C 180,E1 -19917.423,E2 -19917.423} C_VEL
LIN {X 0,Y 250.114,Z 739.654,A -85,B 0,C 180,E1 -19918.88,E2 -19918.88} C_VEL
LIN {X 0,Y 253.174,Z 729.51,A -85,B 0,C 180,E1 -19920.21,E2 -19920.21} C_VEL
LIN {X 0,Y 256.081,Z 717.173,A -85,B 0,C 180,E1 -19921.431,E2 -19921.431} C_VEL
LIN {X 0,Y 258.438,Z 703.236,A -85,B 0,C 180,E1 -19922.429,E2 -19922.429} C_VEL
LIN {X 0,Y 264.58,Z 666.842,A -85,B 0,C 180,E1 -19924.424,E2 -19924.424} C_VEL
LIN {X 0,Y 269.632,Z 638.559,A -85,B 0,C 180,E1 -19925.85,E2 -19925.85} C_VEL
LIN {X 0,Y 270.769,Z 631.998,A -85,B 0,C 180,E1 -19926.309,E2 -19926.309} C_VEL
LIN {X 0,Y 271.611,Z 630.218,A -85,B 0,C 180,E1 -19926.523,E2 -19926.523} C_VEL
LIN {X 0,Y 270.156,Z 628.167,A -85,B 0,C 180,E1 -19928.699,E2 -19928.699} C_VEL
LIN {X 0,Y 269.002,Z 627.157,A -85,B 0,C 180,E1 -19930.781,E2 -19930.781} C_VEL
LIN {X 0,Y 268.111,Z 626.929,A -85,B 0,C 180,E1 -19932.965,E2 -19932.965} C_VEL
LIN {X 0,Y 267.392,Z 627.608,A -85,B 0,C 180,E1 -19935.208,E2 -19935.208} C_VEL
LIN {X 0,Y 266.804,Z 629.336,A -85,B 0,C 180,E1 -19937.526,E2 -19937.526} C_VEL
LIN {X 0,Y 266.2,Z 632.297,A -85,B 0,C 180,E1 -19939.965,E2 -19939.965} C_VEL
LIN {X 0,Y 266.69,Z 636.026,A -85,B 0,C 180,E1 -19941.607,E2 -19941.607} C_VEL
LIN {X 0,Y 266.703,Z 646.243,A -85,B 0,C 180,E1 -19943.549,E2 -19943.549} C_VEL
LIN {X 0,Y 266.905,Z 658.454,A -85,B 0,C 180,E1 -19945.552,E2 -19945.552} C_VEL
LIN {X 0,Y 267.008,Z 671.097,A -85,B 0,C 180,E1 -19947.262,E2 -19947.262} C_VEL
LIN {X 0,Y 267.002,Z 675.318,A -85,B 0,C 180,E1 -19947.755,E2 -19947.755} C_VEL
LIN {X 0,Y 261.299,Z 709.589,A -85,B 0,C 180,E1 -19949.491,E2 -19949.491} C_VEL
LIN {X 0,Y 258.758,Z 721.127,A -85,B 0,C 180,E1 -19950.325,E2 -19950.325} C_VEL
LIN {X 0,Y 255.94,Z 730.78,A -85,B 0,C 180,E1 -19951.279,E2 -19951.279} C_VEL
LIN {X 0,Y 252.368,Z 741.209,A -85,B 0,C 180,E1 -19952.645,E2 -19952.645} C_VEL
LIN {X 0,Y 248.968,Z 749.406,A -85,B 0,C 180,E1 -19954.053,E2 -19954.053} C_VEL
LIN {X 0,Y 245.749,Z 756.256,A -85,B 0,C 180,E1 -19955.501,E2 -19955.501} C_VEL
LIN {X 0,Y 242.17,Z 763.179,A -85,B 0,C 180,E1 -19957.386,E2 -19957.386} C_VEL
LIN {X 0,Y 238.87,Z 768.608,A -85,B 0,C 180,E1 -19959.325,E2 -19959.325} C_VEL
LIN {X 0,Y 235.345,Z 773.659,A -85,B 0,C 180,E1 -19961.726,E2 -19961.726} C_VEL
LIN {X 0,Y 232.296,Z 777.278,A -85,B 0,C 180,E1 -19964.199,E2 -19964.199} C_VEL
LIN {X 0,Y 230.693,Z 778.884,A -85,B 0,C 180,E1 -19965.894,E2 -19965.894} C_VEL
LIN {X 0,Y 229.349,Z 779.93,A -85,B 0,C 180,E1 -19967.614,E2 -19967.614} C_VEL
LIN {X 0,Y 228.188,Z 780.448,A -85,B 0,C 180,E1 -19969.351,E2 -19969.351} C_VEL
LIN {X 0,Y 227.316,Z 780.448,A -85,B 0,C 180,E1 -19971.107,E2 -19971.107} C_VEL
LIN {X 0,Y 226.554,Z 779.821,A -85,B 0,C 180,E1 -19973.074,E2 -19973.074} C_VEL
LIN {X 0,Y 226.085,Z 778.863,A -85,B 0,C 180,E1 -19974.649,E2 -19974.649} C_VEL
LIN {X 0,Y 225.831,Z 776.109,A -85,B 0,C 180,E1 -19977.324,E2 -19977.324} C_VEL
LIN {X 0,Y 225.819,Z 772.037,A -85,B 0,C 180,E1 -19980,E2 -19980} C_VEL
LIN {X 0,Y 226.074,Z 766.358,A -85,B 0,C 180,E1 -19982.673,E2 -19982.673} C_VEL
LIN {X 0,Y 226.242,Z 761.414,A -85,B 0,C 180,E1 -19984.454,E2 -19984.454} C_VEL
LIN {X 0,Y 226.557,Z 754.683,A -85,B 0,C 180,E1 -19986.427,E2 -19986.427} C_VEL
LIN {X 0,Y 226.95,Z 746.704,A -85,B 0,C 180,E1 -19988.322,E2 -19988.322} C_VEL
LIN {X 0,Y 227.393,Z 737.638,A -85,B 0,C 180,E1 -19990.012,E2 -19990.012} C_VEL
LIN {X 0,Y 228.013,Z 727.184,A -85,B 0,C 180,E1 -19991.557,E2 -19991.557} C_VEL
LIN {X 0,Y 228.453,Z 715.924,A -85,B 0,C 180,E1 -19992.775,E2 -19992.775} C_VEL
LIN {X 0,Y 228.858,Z 703.757,A -85,B 0,C 180,E1 -19993.712,E2 -19993.712} C_VEL
LIN {X 0,Y 229.97,Z 656.354,A -85,B 0,C 180,E1 -19996.222,E2 -19996.222} C_VEL
LIN {X 0,Y 228.572,Z 634.065,A -85,B 0,C 180,E1 -19997.376,E2 -19997.376} C_VEL
LIN {X 0,Y 228.575,Z 632.179,A -85,B 0,C 180,E1 -19997.521,E2 -19997.521} C_VEL
LIN {X 0,Y 230.088,Z 613.562,A -85,B 0,C 180,E1 -20001.973,E2 -20001.973} C_VEL
LIN {X 0,Y 231.874,Z 594.365,A -85,B 0,C 180,E1 -20006.556,E2 -20006.556} C_VEL
LIN {X 0,Y 233.189,Z 581.769,A -85,B 0,C 180,E1 -20009.547,E2 -20009.547} C_VEL
LIN {X 0,Y 230.563,Z 568.69,A -85,B 0,C 180,E1 -20012.872,E2 -20012.872} C_VEL
LIN {X 0,Y 228.028,Z 556.261,A -85,B 0,C 180,E1 -20016.168,E2 -20016.168} C_VEL
LIN {X 0,Y 227.831,Z 556.072,A -85,B 0,C 180,E1 -20020.376,E2 -20020.376} C_VEL
LIN {X 0,Y 227.855,Z 556.068,A -85,B 0,C 180,E1 -20025.188,E2 -20025.188} C_VEL
LIN {X 0,Y 227.894,Z 556.088,A -85,B 0,C 180,E1 -20027.743,E2 -20027.743} C_VEL
LIN {X 0,Y 227.852,Z 556.072,A -85,B 0,C 180,E1 -20031.909,E2 -20031.909} C_VEL
LIN {X 0,Y 227.907,Z 556.391,A -85,B 0,C 180,E1 -20032.905,E2 -20032.905} C_VEL
LIN {X 0,Y 228.318,Z 557.758,A -85,B 0,C 180,E1 -20033.248,E2 -20033.248} C_VEL
LIN {X 0,Y 232.651,Z 564.974,A -85,B 0,C 180,E1 -20034.328,E2 -20034.328} C_VEL
LIN {X 0,Y 240.566,Z 580.584,A -85,B 0,C 180,E1 -20036.234,E2 -20036.234} C_VEL
LIN {X 0,Y 246.802,Z 594.959,A -85,B 0,C 180,E1 -20037.692,E2 -20037.692} C_VEL
LIN {X 0,Y 248.99,Z 600.601,A -85,B 0,C 180,E1 -20038.201,E2 -20038.201} C_VEL
LIN {X 0,Y 246.577,Z 662.293,A -85,B 0,C 180,E1 -20039.945,E2 -20039.945} C_VEL
LIN {X 0,Y 245.436,Z 675.522,A -85,B 0,C 180,E1 -20040.6,E2 -20040.6} C_VEL
LIN {X 0,Y 243.902,Z 688.683,A -85,B 0,C 180,E1 -20041.61,E2 -20041.61} C_VEL
LIN {X 0,Y 242.133,Z 699.979,A -85,B 0,C 180,E1 -20042.795,E2 -20042.795} C_VEL
LIN {X 0,Y 239.787,Z 711.615,A -85,B 0,C 180,E1 -20044.384,E2 -20044.384} C_VEL
LIN {X 0,Y 237.383,Z 722.382,A -85,B 0,C 180,E1 -20046.278,E2 -20046.278} C_VEL
LIN {X 0,Y 235.311,Z 731.193,A -85,B 0,C 180,E1 -20048.234,E2 -20048.234} C_VEL
LIN {X 0,Y 232.924,Z 739.838,A -85,B 0,C 180,E1 -20050.614,E2 -20050.614} C_VEL
LIN {X 0,Y 230.752,Z 747.242,A -85,B 0,C 180,E1 -20053.18,E2 -20053.18} C_VEL
LIN {X 0,Y 229.049,Z 753.183,A -85,B 0,C 180,E1 -20055.789,E2 -20055.789} C_VEL
LIN {X 0,Y 227.692,Z 757.876,A -85,B 0,C 180,E1 -20058.425,E2 -20058.425} C_VEL
LIN {X 0,Y 226.769,Z 761.46,A -85,B 0,C 180,E1 -20061.084,E2 -20061.084} C_VEL
LIN {X 0,Y 226.109,Z 764.293,A -85,B 0,C 180,E1 -20064.066,E2 -20064.066} C_VEL
LIN {X 0,Y 225.868,Z 765.693,A -85,B 0,C 180,E1 -20066.431,E2 -20066.431} C_VEL
LIN {X 0,Y 225.748,Z 766.531,A -85,B 0,C 180,E1 -20069.998,E2 -20069.998} C_VEL
LIN {X 0,Y 225.753,Z 766.339,A -85,B 0,C 180,E1 -20071.782,E2 -20071.782} C_VEL
LIN {X 0,Y 225.865,Z 765.754,A -85,B 0,C 180,E1 -20073.566,E2 -20073.566} C_VEL
LIN {X 0,Y 226.332,Z 763.434,A -85,B 0,C 180,E1 -20077.133,E2 -20077.133} C_VEL
LIN {X 0,Y 227.023,Z 760.565,A -85,B 0,C 180,E1 -20079.801,E2 -20079.801} C_VEL
LIN {X 0,Y 228.08,Z 756.673,A -85,B 0,C 180,E1 -20082.455,E2 -20082.455} C_VEL
LIN {X 0,Y 229.54,Z 751.654,A -85,B 0,C 180,E1 -20085.083,E2 -20085.083} C_VEL
LIN {X 0,Y 231.317,Z 745.333,A -85,B 0,C 180,E1 -20087.686,E2 -20087.686} C_VEL
LIN {X 0,Y 233.696,Z 737.413,A -85,B 0,C 180,E1 -20090.231,E2 -20090.231} C_VEL
LIN {X 0,Y 235.716,Z 729.67,A -85,B 0,C 180,E1 -20092.257,E2 -20092.257} C_VEL
LIN {X 0,Y 238.101,Z 719.498,A -85,B 0,C 180,E1 -20094.406,E2 -20094.406} C_VEL
LIN {X 0,Y 240.515,Z 708.409,A -85,B 0,C 180,E1 -20096.227,E2 -20096.227} C_VEL
LIN {X 0,Y 242.592,Z 697.529,A -85,B 0,C 180,E1 -20097.613,E2 -20097.613} C_VEL
LIN {X 0,Y 244.444,Z 685.495,A -85,B 0,C 180,E1 -20098.787,E2 -20098.787} C_VEL
LIN {X 0,Y 245.828,Z 673.301,A -85,B 0,C 180,E1 -20099.652,E2 -20099.652} C_VEL
LIN {X 0,Y 246.802,Z 660.96,A -85,B 0,C 180,E1 -20100.214,E2 -20100.214} C_VEL
LIN {X 0,Y 248.948,Z 600.444,A -85,B 0,C 180,E1 -20101.947,E2 -20101.947} C_VEL
LIN {X 0,Y 243.131,Z 586.222,A -85,B 0,C 180,E1 -20103.304,E2 -20103.304} C_VEL
LIN {X 0,Y 235.849,Z 571.019,A -85,B 0,C 180,E1 -20105.036,E2 -20105.036} C_VEL
LIN {X 0,Y 229.88,Z 560.166,A -85,B 0,C 180,E1 -20106.506,E2 -20106.506} C_VEL
LIN {X 0,Y 228.41,Z 558.012,A -85,B 0,C 180,E1 -20106.869,E2 -20106.869} C_VEL
LIN {X 0,Y 227.89,Z 556.226,A -85,B 0,C 180,E1 -20107.183,E2 -20107.183} C_VEL
LIN {X 0,Y 227.83,Z 556.091,A -85,B 0,C 180,E1 -20110.373,E2 -20110.373} C_VEL
LIN {X 0,Y 227.832,Z 556.082,A -85,B 0,C 180,E1 -20115.191,E2 -20115.191} C_VEL
LIN {X 0,Y 227.869,Z 556.08,A -85,B 0,C 180,E1 -20119.632,E2 -20119.632} C_VEL
LIN {X 0,Y 227.896,Z 556.09,A -85,B 0,C 180,E1 -20124.131,E2 -20124.131} C_VEL
LIN {X 0,Y 227.868,Z 556.094,A -85,B 0,C 180,E1 -20128.377,E2 -20128.377} C_VEL
LIN {X 0,Y 227.88,Z 556.085,A -85,B 0,C 180,E1 -20132.444,E2 -20132.444} C_VEL
LIN {X 0,Y 227.908,Z 556.09,A -85,B 0,C 180,E1 -20136.367,E2 -20136.367} C_VEL
LIN {X 0,Y 227.936,Z 556.091,A -85,B 0,C 180,E1 -20140.174,E2 -20140.174} C_VEL
LIN {X 0,Y 228.051,Z 556.06,A -85,B 0,C 180,E1 -20143.897,E2 -20143.897} C_VEL
LIN {X 0,Y 228.087,Z 556.071,A -85,B 0,C 180,E1 -20147.544,E2 -20147.544} C_VEL
LIN {X 0,Y 228.299,Z 556.031,A -85,B 0,C 180,E1 -20151.146,E2 -20151.146} C_VEL
LIN {X 0,Y 228.349,Z 556.039,A -85,B 0,C 180,E1 -20152.928,E2 -20152.928} C_VEL
LIN {X 0,Y 228.549,Z 556.003,A -85,B 0,C 180,E1 -20158.238,E2 -20158.238} C_VEL
LIN {X 0,Y 228.549,Z 556.009,A -85,B 0,C 180,E1 -20161.762,E2 -20161.762} C_VEL
LIN {X 0,Y 228.352,Z 556.04,A -85,B 0,C 180,E1 -20167.071,E2 -20167.071} C_VEL
LIN {X 0,Y 228.165,Z 556.046,A -85,B 0,C 180,E1 -20170.65,E2 -20170.65} C_VEL
LIN {X 0,Y 228.087,Z 556.064,A -85,B 0,C 180,E1 -20171.94,E2 -20171.94} C_VEL
LIN {X 0,Y 227.392,Z 556.163,A -85,B 0,C 180,E1 -20173.414,E2 -20173.414} C_VEL
LIN {X 0,Y 224.47,Z 556.53,A -85,B 0,C 180,E1 -20175.818,E2 -20175.818} C_VEL
LIN {X 0,Y 221.999,Z 556.829,A -85,B 0,C 180,E1 -20177.78,E2 -20177.78} C_VEL
LIN {X 0,Y 220.949,Z 556.964,A -85,B 0,C 180,E1 -20179.305,E2 -20179.305} C_VEL
LIN {X 0,Y 220.868,Z 556.964,A -85,B 0,C 180,E1 -20179.822,E2 -20179.822} C_VEL
LIN {X 0,Y 220.861,Z 556.974,A -85,B 0,C 180,E1 -20184.436,E2 -20184.436} C_VEL
LIN {X 0,Y 220.821,Z 556.979,A -85,B 0,C 180,E1 -20188.516,E2 -20188.516} C_VEL
LIN {X 0,Y 220.81,Z 556.98,A -85,B 0,C 180,E1 -20192.757,E2 -20192.757} C_VEL
LIN {X 0,Y 220.833,Z 556.948,A -85,B 0,C 180,E1 -20197.289,E2 -20197.289} C_VEL
LIN {X 0,Y 220.814,Z 556.959,A -85,B 0,C 180,E1 -20201.942,E2 -20201.942} C_VEL
LIN {X 0,Y 220.869,Z 557.068,A -85,B 0,C 180,E1 -20207.042,E2 -20207.042} C_VEL
LIN {X 0,Y 222.873,Z 564.567,A -85,B 0,C 180,E1 -20211.174,E2 -20211.174} C_VEL
LIN {X 0,Y 223.4,Z 566.701,A -85,B 0,C 180,E1 -20212.093,E2 -20212.093} C_VEL
LIN {X 0,Y 230.121,Z 580.028,A -85,B 0,C 180,E1 -20213.931,E2 -20213.931} C_VEL
LIN {X 0,Y 237.565,Z 596.707,A -85,B 0,C 180,E1 -20215.818,E2 -20215.818} C_VEL
LIN {X 0,Y 239.8,Z 602.532,A -85,B 0,C 180,E1 -20216.383,E2 -20216.383} C_VEL
LIN {X 0,Y 242.343,Z 621.659,A -85,B 0,C 180,E1 -20217.438,E2 -20217.438} C_VEL
LIN {X 0,Y 240.041,Z 675.899,A -85,B 0,C 180,E1 -20219.024,E2 -20219.024} C_VEL
LIN {X 0,Y 238.723,Z 689.343,A -85,B 0,C 180,E1 -20219.732,E2 -20219.732} C_VEL
LIN {X 0,Y 236.911,Z 701.7,A -85,B 0,C 180,E1 -20220.696,E2 -20220.696} C_VEL
LIN {X 0,Y 234.615,Z 714.386,A -85,B 0,C 180,E1 -20222.094,E2 -20222.094} C_VEL
LIN {X 0,Y 232.116,Z 725.657,A -85,B 0,C 180,E1 -20223.718,E2 -20223.718} C_VEL
LIN {X 0,Y 229.56,Z 735.813,A -85,B 0,C 180,E1 -20225.589,E2 -20225.589} C_VEL
LIN {X 0,Y 227.119,Z 744.969,A -85,B 0,C 180,E1 -20227.726,E2 -20227.726} C_VEL
LIN {X 0,Y 224.714,Z 753.898,A -85,B 0,C 180,E1 -20230.356,E2 -20230.356} C_VEL
LIN {X 0,Y 222.584,Z 761.082,A -85,B 0,C 180,E1 -20233.02,E2 -20233.02} C_VEL
LIN {X 0,Y 220.622,Z 767.623,A -85,B 0,C 180,E1 -20236.179,E2 -20236.179} C_VEL
LIN {X 0,Y 219.595,Z 771.962,A -85,B 0,C 180,E1 -20238.931,E2 -20238.931} C_VEL
LIN {X 0,Y 219.091,Z 774.263,A -85,B 0,C 180,E1 -20240.772,E2 -20240.772} C_VEL
LIN {X 0,Y 218.759,Z 776.126,A -85,B 0,C 180,E1 -20242.618,E2 -20242.618} C_VEL
LIN {X 0,Y 218.481,Z 778.255,A -85,B 0,C 180,E1 -20245.71,E2 -20245.71} C_VEL
LIN {X 0,Y 218.538,Z 779.131,A -85,B 0,C 180,E1 -20248.159,E2 -20248.159} C_VEL
LIN {X 0,Y 218.612,Z 779.344,A -85,B 0,C 180,E1 -20250.002,E2 -20250.002} C_VEL
LIN {X 0,Y 218.766,Z 778.835,A -85,B 0,C 180,E1 -20253.224,E2 -20253.224} C_VEL
LIN {X 0,Y 218.818,Z 781.128,A -85,B 0,C 180,E1 -20255.531,E2 -20255.531} C_VEL
LIN {X 0,Y 219.067,Z 782.385,A -85,B 0,C 180,E1 -20257.374,E2 -20257.374} C_VEL
LIN {X 0,Y 219.508,Z 783.117,A -85,B 0,C 180,E1 -20259.213,E2 -20259.213} C_VEL
LIN {X 0,Y 220.263,Z 783.345,A -85,B 0,C 180,E1 -20261.039,E2 -20261.039} C_VEL
LIN {X 0,Y 221.273,Z 782.997,A -85,B 0,C 180,E1 -20262.848,E2 -20262.848} C_VEL
LIN {X 0,Y 222.46,Z 782.103,A -85,B 0,C 180,E1 -20264.641,E2 -20264.641} C_VEL
LIN {X 0,Y 223.886,Z 780.722,A -85,B 0,C 180,E1 -20266.412,E2 -20266.412} C_VEL
LIN {X 0,Y 226.532,Z 777.657,A -85,B 0,C 180,E1 -20269.013,E2 -20269.013} C_VEL
LIN {X 0,Y 229.798,Z 773.256,A -85,B 0,C 180,E1 -20271.532,E2 -20271.532} C_VEL
LIN {X 0,Y 232.858,Z 768.406,A -85,B 0,C 180,E1 -20273.574,E2 -20273.574} C_VEL
LIN {X 0,Y 236.186,Z 762.386,A -85,B 0,C 180,E1 -20275.562,E2 -20275.562} C_VEL
LIN {X 0,Y 239.858,Z 755.103,A -85,B 0,C 180,E1 -20277.484,E2 -20277.484} C_VEL
LIN {X 0,Y 243.822,Z 745.767,A -85,B 0,C 180,E1 -20279.343,E2 -20279.343} C_VEL
LIN {X 0,Y 247.746,Z 735.362,A -85,B 0,C 180,E1 -20280.943,E2 -20280.943} C_VEL
LIN {X 0,Y 250.868,Z 724.857,A -85,B 0,C 180,E1 -20282.161,E2 -20282.161} C_VEL
LIN {X 0,Y 253.67,Z 712.802,A -85,B 0,C 180,E1 -20283.234,E2 -20283.234} C_VEL
LIN {X 0,Y 256.711,Z 695.572,A -85,B 0,C 180,E1 -20284.32,E2 -20284.32} C_VEL
LIN {X 0,Y 262.09,Z 666.43,A -85,B 0,C 180,E1 -20285.887,E2 -20285.887} C_VEL
LIN {X 0,Y 267.235,Z 639.496,A -85,B 0,C 180,E1 -20287.265,E2 -20287.265} C_VEL
LIN {X 0,Y 267.838,Z 635.695,A -85,B 0,C 180,E1 -20287.528,E2 -20287.528} C_VEL
LIN {X 0,Y 266.347,Z 634.102,A -85,B 0,C 180,E1 -20289.129,E2 -20289.129} C_VEL
LIN {X 0,Y 264.493,Z 632.879,A -85,B 0,C 180,E1 -20291.926,E2 -20291.926} C_VEL
LIN {X 0,Y 263.587,Z 633.26,A -85,B 0,C 180,E1 -20294.649,E2 -20294.649} C_VEL
LIN {X 0,Y 263.451,Z 635.581,A -85,B 0,C 180,E1 -20297.338,E2 -20297.338} C_VEL
LIN {X 0,Y 264.025,Z 639.067,A -85,B 0,C 180,E1 -20299.687,E2 -20299.687} C_VEL
LIN {X 0,Y 264.352,Z 641.834,A -85,B 0,C 180,E1 -20300.83,E2 -20300.83} C_VEL
LIN {X 0,Y 263.932,Z 655.214,A -85,B 0,C 180,E1 -20303.299,E2 -20303.299} C_VEL
LIN {X 0,Y 263.743,Z 666.414,A -85,B 0,C 180,E1 -20305.045,E2 -20305.045} C_VEL
LIN {X 0,Y 263.553,Z 677.153,A -85,B 0,C 180,E1 -20306.455,E2 -20306.455} C_VEL
LIN {X 0,Y 257.667,Z 710.343,A -85,B 0,C 180,E1 -20308.156,E2 -20308.156} C_VEL
LIN {X 0,Y 254.81,Z 722.073,A -85,B 0,C 180,E1 -20309.031,E2 -20309.031} C_VEL
LIN {X 0,Y 251.664,Z 731.945,A -85,B 0,C 180,E1 -20310.031,E2 -20310.031} C_VEL
LIN {X 0,Y 247.826,Z 742.177,A -85,B 0,C 180,E1 -20311.409,E2 -20311.409} C_VEL
LIN {X 0,Y 244.663,Z 749.316,A -85,B 0,C 180,E1 -20312.638,E2 -20312.638} C_VEL
LIN {X 0,Y 241.214,Z 756.115,A -85,B 0,C 180,E1 -20314.085,E2 -20314.085} C_VEL
LIN {X 0,Y 237.307,Z 763.063,A -85,B 0,C 180,E1 -20315.97,E2 -20315.97} C_VEL
LIN {X 0,Y 233.764,Z 768.533,A -85,B 0,C 180,E1 -20317.926,E2 -20317.926} C_VEL
LIN {X 0,Y 229.873,Z 773.565,A -85,B 0,C 180,E1 -20320.348,E2 -20320.348} C_VEL
LIN {X 0,Y 227.556,Z 776.126,A -85,B 0,C 180,E1 -20322.01,E2 -20322.01} C_VEL
LIN {X 0,Y 225.523,Z 778.088,A -85,B 0,C 180,E1 -20323.712,E2 -20323.712} C_VEL
LIN {X 0,Y 223.849,Z 779.483,A -85,B 0,C 180,E1 -20325.453,E2 -20325.453} C_VEL
LIN {X 0,Y 222.452,Z 780.346,A -85,B 0,C 180,E1 -20327.223,E2 -20327.223} C_VEL
LIN {X 0,Y 221.22,Z 780.644,A -85,B 0,C 180,E1 -20329.011,E2 -20329.011} C_VEL
LIN {X 0,Y 220.304,Z 780.375,A -85,B 0,C 180,E1 -20330.822,E2 -20330.822} C_VEL
LIN {X 0,Y 219.347,Z 779.203,A -85,B 0,C 180,E1 -20333.353,E2 -20333.353} C_VEL
LIN {X 0,Y 218.862,Z 776.463,A -85,B 0,C 180,E1 -20336.318,E2 -20336.318} C_VEL
LIN {X 0,Y 218.784,Z 772.479,A -85,B 0,C 180,E1 -20339.08,E2 -20339.08} C_VEL
LIN {X 0,Y 218.98,Z 767.011,A -85,B 0,C 180,E1 -20341.839,E2 -20341.839} C_VEL
LIN {X 0,Y 219.261,Z 760.901,A -85,B 0,C 180,E1 -20344.136,E2 -20344.136} C_VEL
LIN {X 0,Y 219.541,Z 753.845,A -85,B 0,C 180,E1 -20346.256,E2 -20346.256} C_VEL
LIN {X 0,Y 219.949,Z 745.81,A -85,B 0,C 180,E1 -20348.175,E2 -20348.175} C_VEL
LIN {X 0,Y 220.296,Z 738.118,A -85,B 0,C 180,E1 -20349.642,E2 -20349.642} C_VEL
LIN {X 0,Y 220.918,Z 727.765,A -85,B 0,C 180,E1 -20351.236,E2 -20351.236} C_VEL
LIN {X 0,Y 221.374,Z 716.795,A -85,B 0,C 180,E1 -20352.491,E2 -20352.491} C_VEL
LIN {X 0,Y 221.743,Z 705.071,A -85,B 0,C 180,E1 -20353.46,E2 -20353.46} C_VEL
LIN {X 0,Y 222.851,Z 657.354,A -85,B 0,C 180,E1 -20356.136,E2 -20356.136} C_VEL
LIN {X 0,Y 221.467,Z 633.417,A -85,B 0,C 180,E1 -20357.442,E2 -20357.442} C_VEL
LIN {X 0,Y 221.509,Z 631.894,A -85,B 0,C 180,E1 -20357.609,E2 -20357.609} C_VEL
LIN {X 0,Y 223.07,Z 613.143,A -85,B 0,C 180,E1 -20362.214,E2 -20362.214} C_VEL
LIN {X 0,Y 224.923,Z 593.804,A -85,B 0,C 180,E1 -20366.941,E2 -20366.941} C_VEL
LIN {X 0,Y 226.1,Z 581.969,A -85,B 0,C 180,E1 -20369.824,E2 -20369.824} C_VEL
LIN {X 0,Y 222.485,Z 564.473,A -85,B 0,C 180,E1 -20374.386,E2 -20374.386} C_VEL
LIN {X 0,Y 220.973,Z 557.135,A -85,B 0,C 180,E1 -20376.431,E2 -20376.431} C_VEL
LIN {X 0,Y 220.8,Z 556.949,A -85,B 0,C 180,E1 -20380.188,E2 -20380.188} C_VEL
LIN {X 0,Y 220.787,Z 556.934,A -85,B 0,C 180,E1 -20384.451,E2 -20384.451} C_VEL
LIN {X 0,Y 220.836,Z 556.959,A -85,B 0,C 180,E1 -20388.061,E2 -20388.061} C_VEL
LIN {X 0,Y 220.828,Z 557.072,A -85,B 0,C 180,E1 -20391.366,E2 -20391.366} C_VEL
LIN {X 0,Y 221.047,Z 558.04,A -85,B 0,C 180,E1 -20391.802,E2 -20391.802} C_VEL
LIN {X 0,Y 222.664,Z 560.956,A -85,B 0,C 180,E1 -20392.285,E2 -20392.285} C_VEL
LIN {X 0,Y 226.717,Z 567.452,A -85,B 0,C 180,E1 -20393.331,E2 -20393.331} C_VEL
LIN {X 0,Y 233.118,Z 579.651,A -85,B 0,C 180,E1 -20394.956,E2 -20394.956} C_VEL
LIN {X 0,Y 239.682,Z 594.161,A -85,B 0,C 180,E1 -20396.571,E2 -20396.571} C_VEL
LIN {X 0,Y 242.854,Z 602.191,A -85,B 0,C 180,E1 -20397.345,E2 -20397.345} C_VEL
LIN {X 0,Y 240.495,Z 662.171,A -85,B 0,C 180,E1 -20399.088,E2 -20399.088} C_VEL
LIN {X 0,Y 239.347,Z 675.185,A -85,B 0,C 180,E1 -20399.731,E2 -20399.731} C_VEL
LIN {X 0,Y 237.872,Z 687.767,A -85,B 0,C 180,E1 -20400.701,E2 -20400.701} C_VEL
LIN {X 0,Y 236.17,Z 698.457,A -85,B 0,C 180,E1 -20401.808,E2 -20401.808} C_VEL
LIN {X 0,Y 233.984,Z 709.195,A -85,B 0,C 180,E1 -20403.22,E2 -20403.22} C_VEL
LIN {X 0,Y 231.464,Z 720.14,A -85,B 0,C 180,E1 -20405.082,E2 -20405.082} C_VEL
LIN {X 0,Y 228.849,Z 730.664,A -85,B 0,C 180,E1 -20407.388,E2 -20407.388} C_VEL
LIN {X 0,Y 226.665,Z 738.659,A -85,B 0,C 180,E1 -20409.583,E2 -20409.583} C_VEL
LIN {X 0,Y 224.32,Z 746.339,A -85,B 0,C 180,E1 -20412.212,E2 -20412.212} C_VEL
LIN {X 0,Y 222.172,Z 753.389,A -85,B 0,C 180,E1 -20415.339,E2 -20415.339} C_VEL
LIN {X 0,Y 220.725,Z 758.083,A -85,B 0,C 180,E1 -20418.054,E2 -20418.054} C_VEL
LIN {X 0,Y 219.767,Z 761.665,A -85,B 0,C 180,E1 -20420.798,E2 -20420.798} C_VEL
LIN {X 0,Y 219.001,Z 764.723,A -85,B 0,C 180,E1 -20424.173,E2 -20424.173} C_VEL
LIN {X 0,Y 218.779,Z 765.898,A -85,B 0,C 180,E1 -20426.315,E2 -20426.315} C_VEL
LIN {X 0,Y 218.674,Z 766.507,A -85,B 0,C 180,E1 -20428.157,E2 -20428.157} C_VEL
LIN {X 0,Y 218.663,Z 766.735,A -85,B 0,C 180,E1 -20429.998,E2 -20429.998} C_VEL
LIN {X 0,Y 218.673,Z 766.543,A -85,B 0,C 180,E1 -20431.84,E2 -20431.84} C_VEL
LIN {X 0,Y 218.776,Z 765.958,A -85,B 0,C 180,E1 -20433.682,E2 -20433.682} C_VEL
LIN {X 0,Y 219,Z 764.813,A -85,B 0,C 180,E1 -20435.824,E2 -20435.824} C_VEL
LIN {X 0,Y 219.765,Z 761.824,A -85,B 0,C 180,E1 -20439.199,E2 -20439.199} C_VEL
LIN {X 0,Y 220.709,Z 758.291,A -85,B 0,C 180,E1 -20441.944,E2 -20441.944} C_VEL
LIN {X 0,Y 222.125,Z 753.655,A -85,B 0,C 180,E1 -20444.66,E2 -20444.66} C_VEL
LIN {X 0,Y 224.205,Z 746.669,A -85,B 0,C 180,E1 -20447.794,E2 -20447.794} C_VEL
LIN {X 0,Y 226.611,Z 739.086,A -85,B 0,C 180,E1 -20450.418,E2 -20450.418} C_VEL
LIN {X 0,Y 228.985,Z 730.514,A -85,B 0,C 180,E1 -20452.775,E2 -20452.775} C_VEL
LIN {X 0,Y 231.377,Z 720.765,A -85,B 0,C 180,E1 -20454.924,E2 -20454.924} C_VEL
LIN {X 0,Y 233.905,Z 710.002,A -85,B 0,C 180,E1 -20456.786,E2 -20456.786} C_VEL
LIN {X 0,Y 236.04,Z 699.49,A -85,B 0,C 180,E1 -20458.206,E2 -20458.206} C_VEL
LIN {X 0,Y 238.058,Z 686.82,A -85,B 0,C 180,E1 -20459.513,E2 -20459.513} C_VEL
LIN {X 0,Y 239.673,Z 673.756,A -85,B 0,C 180,E1 -20460.474,E2 -20460.474} C_VEL
LIN {X 0,Y 240.716,Z 660.771,A -85,B 0,C 180,E1 -20461.076,E2 -20461.076} C_VEL
LIN {X 0,Y 242.963,Z 602.404,A -85,B 0,C 180,E1 -20462.77,E2 -20462.77} C_VEL
LIN {X 0,Y 237.074,Z 588.166,A -85,B 0,C 180,E1 -20464.208,E2 -20464.208} C_VEL
LIN {X 0,Y 229.283,Z 572.038,A -85,B 0,C 180,E1 -20466.163,E2 -20466.163} C_VEL
LIN {X 0,Y 224.945,Z 564.528,A -85,B 0,C 180,E1 -20467.276,E2 -20467.276} C_VEL
LIN {X 0,Y 222.775,Z 561.036,A -85,B 0,C 180,E1 -20467.845,E2 -20467.845} C_VEL
LIN {X 0,Y 221.227,Z 558.589,A -85,B 0,C 180,E1 -20468.258,E2 -20468.258} C_VEL
LIN {X 0,Y 220.816,Z 556.984,A -85,B 0,C 180,E1 -20468.5,E2 -20468.5} C_VEL
LIN {X 0,Y 220.766,Z 556.978,A -85,B 0,C 180,E1 -20472.929,E2 -20472.929} C_VEL
LIN {X 0,Y 220.805,Z 556.975,A -85,B 0,C 180,E1 -20477.057,E2 -20477.057} C_VEL
LIN {X 0,Y 220.845,Z 556.944,A -85,B 0,C 180,E1 -20480.471,E2 -20480.471} C_VEL
LIN {X 0,Y 220.811,Z 556.981,A -85,B 0,C 180,E1 -20485.047,E2 -20485.047} C_VEL
LIN {X 0,Y 220.863,Z 556.973,A -85,B 0,C 180,E1 -20489.394,E2 -20489.394} C_VEL
LIN {X 0,Y 220.89,Z 556.961,A -85,B 0,C 180,E1 -20493.549,E2 -20493.549} C_VEL
LIN {X 0,Y 220.872,Z 556.956,A -85,B 0,C 180,E1 -20497.553,E2 -20497.553} C_VEL
LIN {X 0,Y 220.978,Z 556.946,A -85,B 0,C 180,E1 -20502.57,E2 -20502.57} C_VEL
LIN {X 0,Y 221.02,Z 556.954,A -85,B 0,C 180,E1 -20507.139,E2 -20507.139} C_VEL
LIN {X 0,Y 221.23,Z 556.909,A -85,B 0,C 180,E1 -20510.86,E2 -20510.86} C_VEL
LIN {X 0,Y 221.3,Z 556.917,A -85,B 0,C 180,E1 -20512.702,E2 -20512.702} C_VEL
LIN {X 0,Y 221.506,Z 556.879,A -85,B 0,C 180,E1 -20518.182,E2 -20518.182} C_VEL
LIN {X 0,Y 221.507,Z 556.885,A -85,B 0,C 180,E1 -20521.818,E2 -20521.818} C_VEL
LIN {X 0,Y 221.305,Z 556.919,A -85,B 0,C 180,E1 -20527.298,E2 -20527.298} C_VEL
LIN {X 0,Y 221.11,Z 556.927,A -85,B 0,C 180,E1 -20530.994,E2 -20530.994} C_VEL
LIN {X 0,Y 221.01,Z 556.939,A -85,B 0,C 180,E1 -20536.63,E2 -20536.63} C_VEL
LIN {X 0,Y 220.868,Z 556.964,A -85,B 0,C 180,E1 -20539.822,E2 -20539.822} C_VEL
LIN {X 0,Y 220.225,Z 557.047,A -85,B 0,C 180,E1 -20541.344,E2 -20541.344} C_VEL
LIN {X 0,Y 217.415,Z 557.403,A -85,B 0,C 180,E1 -20543.829,E2 -20543.829} C_VEL
LIN {X 0,Y 214.146,Z 557.801,A -85,B 0,C 180,E1 -20546.901,E2 -20546.901} C_VEL
LIN {X 0,Y 213.78,Z 557.845,A -85,B 0,C 180,E1 -20547.966,E2 -20547.966} C_VEL
LIN {X 0,Y 213.762,Z 557.851,A -85,B 0,C 180,E1 -20551.739,E2 -20551.739} C_VEL
LIN {X 0,Y 213.738,Z 557.829,A -85,B 0,C 180,E1 -20556.29,E2 -20556.29} C_VEL
LIN {X 0,Y 213.75,Z 557.848,A -85,B 0,C 180,E1 -20560.87,E2 -20560.87} C_VEL
LIN {X 0,Y 213.809,Z 557.914,A -85,B 0,C 180,E1 -20565.806,E2 -20565.806} C_VEL
LIN {X 0,Y 215.703,Z 565.1,A -85,B 0,C 180,E1 -20570.011,E2 -20570.011} C_VEL
LIN {X 0,Y 216.135,Z 566.479,A -85,B 0,C 180,E1 -20570.581,E2 -20570.581} C_VEL
LIN {X 0,Y 223.237,Z 580.134,A -85,B 0,C 180,E1 -20572.647,E2 -20572.647} C_VEL
LIN {X 0,Y 230.842,Z 596.808,A -85,B 0,C 180,E1 -20574.689,E2 -20574.689} C_VEL
LIN {X 0,Y 234.061,Z 604.877,A -85,B 0,C 180,E1 -20575.535,E2 -20575.535} C_VEL
LIN {X 0,Y 236.299,Z 621.277,A -85,B 0,C 180,E1 -20576.491,E2 -20576.491} C_VEL
LIN {X 0,Y 234.037,Z 675.099,A -85,B 0,C 180,E1 -20578.103,E2 -20578.103} C_VEL
LIN {X 0,Y 232.708,Z 688.487,A -85,B 0,C 180,E1 -20578.809,E2 -20578.809} C_VEL
LIN {X 0,Y 230.742,Z 701.501,A -85,B 0,C 180,E1 -20579.832,E2 -20579.832} C_VEL
LIN {X 0,Y 228.369,Z 714.186,A -85,B 0,C 180,E1 -20581.261,E2 -20581.261} C_VEL
LIN {X 0,Y 225.764,Z 725.456,A -85,B 0,C 180,E1 -20582.92,E2 -20582.92} C_VEL
LIN {X 0,Y 223.107,Z 735.611,A -85,B 0,C 180,E1 -20584.835,E2 -20584.835} C_VEL
LIN {X 0,Y 220.529,Z 744.766,A -85,B 0,C 180,E1 -20587.023,E2 -20587.023} C_VEL
LIN {X 0,Y 218.02,Z 753.695,A -85,B 0,C 180,E1 -20589.727,E2 -20589.727} C_VEL
LIN {X 0,Y 215.79,Z 760.878,A -85,B 0,C 180,E1 -20592.469,E2 -20592.469} C_VEL
LIN {X 0,Y 213.706,Z 767.419,A -85,B 0,C 180,E1 -20595.723,E2 -20595.723} C_VEL
LIN {X 0,Y 212.599,Z 771.758,A -85,B 0,C 180,E1 -20598.562,E2 -20598.562} C_VEL
LIN {X 0,Y 212.064,Z 774.059,A -85,B 0,C 180,E1 -20600.464,E2 -20600.464} C_VEL
LIN {X 0,Y 211.687,Z 775.921,A -85,B 0,C 180,E1 -20602.37,E2 -20602.37} C_VEL
LIN {X 0,Y 211.393,Z 778.174,A -85,B 0,C 180,E1 -20605.857,E2 -20605.857} C_VEL
LIN {X 0,Y 211.439,Z 778.926,A -85,B 0,C 180,E1 -20608.097,E2 -20608.097} C_VEL
LIN {X 0,Y 211.529,Z 779.14,A -85,B 0,C 180,E1 -20610.002,E2 -20610.002} C_VEL
LIN {X 0,Y 211.739,Z 778.405,A -85,B 0,C 180,E1 -20613.808,E2 -20613.808} C_VEL
LIN {X 0,Y 211.796,Z 780.389,A -85,B 0,C 180,E1 -20615.715,E2 -20615.715} C_VEL
LIN {X 0,Y 212.038,Z 781.887,A -85,B 0,C 180,E1 -20617.62,E2 -20617.62} C_VEL
LIN {X 0,Y 212.509,Z 782.815,A -85,B 0,C 180,E1 -20619.52,E2 -20619.52} C_VEL
LIN {X 0,Y 213.307,Z 783.197,A -85,B 0,C 180,E1 -20621.403,E2 -20621.403} C_VEL
LIN {X 0,Y 214.35,Z 783.083,A -85,B 0,C 180,E1 -20623.27,E2 -20623.27} C_VEL
LIN {X 0,Y 215.598,Z 782.493,A -85,B 0,C 180,E1 -20625.118,E2 -20625.118} C_VEL
LIN {X 0,Y 217.118,Z 781.406,A -85,B 0,C 180,E1 -20626.939,E2 -20626.939} C_VEL
LIN {X 0,Y 219.906,Z 778.694,A -85,B 0,C 180,E1 -20629.609,E2 -20629.609} C_VEL
LIN {X 0,Y 223.36,Z 774.739,A -85,B 0,C 180,E1 -20632.185,E2 -20632.185} C_VEL
LIN {X 0,Y 227.294,Z 769.434,A -85,B 0,C 180,E1 -20634.674,E2 -20634.674} C_VEL
LIN {X 0,Y 230.856,Z 763.737,A -85,B 0,C 180,E1 -20636.684,E2 -20636.684} C_VEL
LIN {X 0,Y 234.794,Z 756.68,A -85,B 0,C 180,E1 -20638.617,E2 -20638.617} C_VEL
LIN {X 0,Y 239.066,Z 748.091,A -85,B 0,C 180,E1 -20640.473,E2 -20640.473} C_VEL
LIN {X 0,Y 242.736,Z 739.329,A -85,B 0,C 180,E1 -20641.899,E2 -20641.899} C_VEL
LIN {X 0,Y 246.203,Z 729.837,A -85,B 0,C 180,E1 -20643.151,E2 -20643.151} C_VEL
LIN {X 0,Y 249.453,Z 718.468,A -85,B 0,C 180,E1 -20644.298,E2 -20644.298} C_VEL
LIN {X 0,Y 252.239,Z 705.53,A -85,B 0,C 180,E1 -20645.245,E2 -20645.245} C_VEL
LIN {X 0,Y 259.54,Z 668.128,A -85,B 0,C 180,E1 -20647.308,E2 -20647.308} C_VEL
LIN {X 0,Y 264.987,Z 641.543,A -85,B 0,C 180,E1 -20648.645,E2 -20648.645} C_VEL
LIN {X 0,Y 263.879,Z 640.436,A -85,B 0,C 180,E1 -20650.004,E2 -20650.004} C_VEL
LIN {X 0,Y 262.685,Z 639.754,A -85,B 0,C 180,E1 -20651.981,E2 -20651.981} C_VEL
LIN {X 0,Y 261.82,Z 640.26,A -85,B 0,C 180,E1 -20654.726,E2 -20654.726} C_VEL
LIN {X 0,Y 261.675,Z 642.497,A -85,B 0,C 180,E1 -20657.188,E2 -20657.188} C_VEL
LIN {X 0,Y 262.018,Z 645.677,A -85,B 0,C 180,E1 -20659.282,E2 -20659.282} C_VEL
LIN {X 0,Y 262.102,Z 647.219,A -85,B 0,C 180,E1 -20659.898,E2 -20659.898} C_VEL
LIN {X 0,Y 261.276,Z 659.85,A -85,B 0,C 180,E1 -20662.272,E2 -20662.272} C_VEL
LIN {X 0,Y 260.747,Z 671.79,A -85,B 0,C 180,E1 -20664.134,E2 -20664.134} C_VEL
LIN {X 0,Y 260.286,Z 679.57,A -85,B 0,C 180,E1 -20665.14,E2 -20665.14} C_VEL
LIN {X 0,Y 254.539,Z 710.093,A -85,B 0,C 180,E1 -20666.708,E2 -20666.708} C_VEL
LIN {X 0,Y 251.622,Z 721.495,A -85,B 0,C 180,E1 -20667.549,E2 -20667.549} C_VEL
LIN {X 0,Y 248.075,Z 731.946,A -85,B 0,C 180,E1 -20668.57,E2 -20668.57} C_VEL
LIN {X 0,Y 243.966,Z 742.3,A -85,B 0,C 180,E1 -20669.965,E2 -20669.965} C_VEL
LIN {X 0,Y 239.901,Z 750.657,A -85,B 0,C 180,E1 -20671.435,E2 -20671.435} C_VEL
LIN {X 0,Y 235.156,Z 759.14,A -85,B 0,C 180,E1 -20673.365,E2 -20673.365} C_VEL
LIN {X 0,Y 231.078,Z 765.374,A -85,B 0,C 180,E1 -20675.279,E2 -20675.279} C_VEL
LIN {X 0,Y 227.367,Z 770.348,A -85,B 0,C 180,E1 -20677.271,E2 -20677.271} C_VEL
LIN {X 0,Y 223.338,Z 774.994,A -85,B 0,C 180,E1 -20679.748,E2 -20679.748} C_VEL
LIN {X 0,Y 220.899,Z 777.251,A -85,B 0,C 180,E1 -20681.449,E2 -20681.449} C_VEL
LIN {X 0,Y 218.771,Z 778.883,A -85,B 0,C 180,E1 -20683.194,E2 -20683.194} C_VEL
LIN {X 0,Y 217.026,Z 779.982,A -85,B 0,C 180,E1 -20684.985,E2 -20684.985} C_VEL
LIN {X 0,Y 215.534,Z 780.57,A -85,B 0,C 180,E1 -20686.806,E2 -20686.806} C_VEL
LIN {X 0,Y 214.277,Z 780.656,A -85,B 0,C 180,E1 -20688.651,E2 -20688.651} C_VEL
LIN {X 0,Y 213.306,Z 780.237,A -85,B 0,C 180,E1 -20690.518,E2 -20690.518} C_VEL
LIN {X 0,Y 212.234,Z 778.417,A -85,B 0,C 180,E1 -20693.44,E2 -20693.44} C_VEL
LIN {X 0,Y 211.833,Z 775.569,A -85,B 0,C 180,E1 -20696.195,E2 -20696.195} C_VEL
LIN {X 0,Y 211.768,Z 771.345,A -85,B 0,C 180,E1 -20699.049,E2 -20699.049} C_VEL
LIN {X 0,Y 211.949,Z 766.499,A -85,B 0,C 180,E1 -20701.425,E2 -20701.425} C_VEL
LIN {X 0,Y 212.214,Z 761.671,A -85,B 0,C 180,E1 -20703.323,E2 -20703.323} C_VEL
LIN {X 0,Y 212.466,Z 754.108,A -85,B 0,C 180,E1 -20705.695,E2 -20705.695} C_VEL
LIN {X 0,Y 212.886,Z 746.658,A -85,B 0,C 180,E1 -20707.588,E2 -20707.588} C_VEL
LIN {X 0,Y 213.253,Z 738.597,A -85,B 0,C 180,E1 -20709.221,E2 -20709.221} C_VEL
LIN {X 0,Y 213.783,Z 728.271,A -85,B 0,C 180,E1 -20710.896,E2 -20710.896} C_VEL
LIN {X 0,Y 214.27,Z 717.643,A -85,B 0,C 180,E1 -20712.19,E2 -20712.19} C_VEL
LIN {X 0,Y 214.668,Z 705.454,A -85,B 0,C 180,E1 -20713.249,E2 -20713.249} C_VEL
LIN {X 0,Y 215.756,Z 657.172,A -85,B 0,C 180,E1 -20716.074,E2 -20716.074} C_VEL
LIN {X 0,Y 214.376,Z 634.007,A -85,B 0,C 180,E1 -20717.397,E2 -20717.397} C_VEL
LIN {X 0,Y 214.409,Z 632.127,A -85,B 0,C 180,E1 -20717.564,E2 -20717.564} C_VEL
LIN {X 0,Y 216.038,Z 612.608,A -85,B 0,C 180,E1 -20722.473,E2 -20722.473} C_VEL
LIN {X 0,Y 217.973,Z 593.129,A -85,B 0,C 180,E1 -20727.352,E2 -20727.352} C_VEL
LIN {X 0,Y 219.014,Z 582.721,A -85,B 0,C 180,E1 -20729.954,E2 -20729.954} C_VEL
LIN {X 0,Y 215.612,Z 566.154,A -85,B 0,C 180,E1 -20734.378,E2 -20734.378} C_VEL
LIN {X 0,Y 213.922,Z 558.002,A -85,B 0,C 180,E1 -20736.683,E2 -20736.683} C_VEL
LIN {X 0,Y 213.717,Z 557.813,A -85,B 0,C 180,E1 -20741.124,E2 -20741.124} C_VEL
LIN {X 0,Y 213.781,Z 557.844,A -85,B 0,C 180,E1 -20746.339,E2 -20746.339} C_VEL
LIN {X 0,Y 213.805,Z 557.997,A -85,B 0,C 180,E1 -20749.96,E2 -20749.96} C_VEL
LIN {X 0,Y 214.076,Z 559.145,A -85,B 0,C 180,E1 -20750.371,E2 -20750.371} C_VEL
LIN {X 0,Y 215.735,Z 561.902,A -85,B 0,C 180,E1 -20750.875,E2 -20750.875} C_VEL
LIN {X 0,Y 216.647,Z 563.247,A -85,B 0,C 180,E1 -20751.129,E2 -20751.129} C_VEL
LIN {X 0,Y 222.791,Z 573.225,A -85,B 0,C 180,E1 -20752.799,E2 -20752.799} C_VEL
LIN {X 0,Y 230.634,Z 589.039,A -85,B 0,C 180,E1 -20754.87,E2 -20754.87} C_VEL
LIN {X 0,Y 236.854,Z 604.113,A -85,B 0,C 180,E1 -20756.471,E2 -20756.471} C_VEL
LIN {X 0,Y 234.406,Z 663.199,A -85,B 0,C 180,E1 -20758.232,E2 -20758.232} C_VEL
LIN {X 0,Y 233.172,Z 676.185,A -85,B 0,C 180,E1 -20758.907,E2 -20758.907} C_VEL
LIN {X 0,Y 231.541,Z 689.106,A -85,B 0,C 180,E1 -20759.944,E2 -20759.944} C_VEL
LIN {X 0,Y 229.641,Z 700.398,A -85,B 0,C 180,E1 -20761.181,E2 -20761.181} C_VEL
LIN {X 0,Y 227.068,Z 712.033,A -85,B 0,C 180,E1 -20762.835,E2 -20762.835} C_VEL
LIN {X 0,Y 224.507,Z 722.479,A -85,B 0,C 180,E1 -20764.752,E2 -20764.752} C_VEL
LIN {X 0,Y 221.998,Z 732.163,A -85,B 0,C 180,E1 -20767.019,E2 -20767.019} C_VEL
LIN {X 0,Y 219.59,Z 740.252,A -85,B 0,C 180,E1 -20769.385,E2 -20769.385} C_VEL
LIN {X 0,Y 217.21,Z 747.655,A -85,B 0,C 180,E1 -20772.097,E2 -20772.097} C_VEL
LIN {X 0,Y 215.316,Z 753.596,A -85,B 0,C 180,E1 -20774.862,E2 -20774.862} C_VEL
LIN {X 0,Y 213.78,Z 758.289,A -85,B 0,C 180,E1 -20777.66,E2 -20777.66} C_VEL
LIN {X 0,Y 212.74,Z 761.871,A -85,B 0,C 180,E1 -20780.491,E2 -20780.491} C_VEL
LIN {X 0,Y 212.244,Z 763.722,A -85,B 0,C 180,E1 -20782.387,E2 -20782.387} C_VEL
LIN {X 0,Y 211.893,Z 765.113,A -85,B 0,C 180,E1 -20784.288,E2 -20784.288} C_VEL
LIN {X 0,Y 211.694,Z 766.103,A -85,B 0,C 180,E1 -20786.191,E2 -20786.191} C_VEL
LIN {X 0,Y 211.596,Z 766.711,A -85,B 0,C 180,E1 -20788.095,E2 -20788.095} C_VEL
LIN {X 0,Y 211.58,Z 766.939,A -85,B 0,C 180,E1 -20789.998,E2 -20789.998} C_VEL
LIN {X 0,Y 211.595,Z 766.747,A -85,B 0,C 180,E1 -20791.902,E2 -20791.902} C_VEL
LIN {X 0,Y 211.692,Z 766.163,A -85,B 0,C 180,E1 -20793.805,E2 -20793.805} C_VEL
LIN {X 0,Y 212.242,Z 763.842,A -85,B 0,C 180,E1 -20797.61,E2 -20797.61} C_VEL
LIN {X 0,Y 213.016,Z 760.973,A -85,B 0,C 180,E1 -20800.453,E2 -20800.453} C_VEL
LIN {X 0,Y 214.206,Z 757.08,A -85,B 0,C 180,E1 -20803.276,E2 -20803.276} C_VEL
LIN {X 0,Y 215.861,Z 752.06,A -85,B 0,C 180,E1 -20806.064,E2 -20806.064} C_VEL
LIN {X 0,Y 217.856,Z 745.738,A -85,B 0,C 180,E1 -20808.818,E2 -20808.818} C_VEL
LIN {X 0,Y 220.444,Z 737.817,A -85,B 0,C 180,E1 -20811.506,E2 -20811.506} C_VEL
LIN {X 0,Y 222.832,Z 729.264,A -85,B 0,C 180,E1 -20813.844,E2 -20813.844} C_VEL
LIN {X 0,Y 225.254,Z 719.9,A -85,B 0,C 180,E1 -20815.898,E2 -20815.898} C_VEL
LIN {X 0,Y 227.883,Z 708.808,A -85,B 0,C 180,E1 -20817.803,E2 -20817.803} C_VEL
LIN {X 0,Y 230.142,Z 697.925,A -85,B 0,C 180,E1 -20819.247,E2 -20819.247} C_VEL
LIN {X 0,Y 232.117,Z 685.888,A -85,B 0,C 180,E1 -20820.472,E2 -20820.472} C_VEL
LIN {X 0,Y 233.666,Z 673.45,A -85,B 0,C 180,E1 -20821.382,E2 -20821.382} C_VEL
LIN {X 0,Y 234.684,Z 660.7,A -85,B 0,C 180,E1 -20821.979,E2 -20821.979} C_VEL
LIN {X 0,Y 236.969,Z 604.268,A -85,B 0,C 180,E1 -20823.648,E2 -20823.648} C_VEL
LIN {X 0,Y 231.162,Z 590.239,A -85,B 0,C 180,E1 -20825.14,E2 -20825.14} C_VEL
LIN {X 0,Y 222.896,Z 573.331,A -85,B 0,C 180,E1 -20827.329,E2 -20827.329} C_VEL
LIN {X 0,Y 217.792,Z 565.182,A -85,B 0,C 180,E1 -20828.705,E2 -20828.705} C_VEL
LIN {X 0,Y 216.004,Z 562.204,A -85,B 0,C 180,E1 -20829.213,E2 -20829.213} C_VEL
LIN {X 0,Y 214.284,Z 559.764,A -85,B 0,C 180,E1 -20829.697,E2 -20829.697} C_VEL
LIN {X 0,Y 213.763,Z 557.841,A -85,B 0,C 180,E1 -20829.951,E2 -20829.951} C_VEL
LIN {X 0,Y 213.704,Z 557.847,A -85,B 0,C 180,E1 -20833.676,E2 -20833.676} C_VEL
LIN {X 0,Y 213.743,Z 557.843,A -85,B 0,C 180,E1 -20836.331,E2 -20836.331} C_VEL
LIN {X 0,Y 213.758,Z 557.844,A -85,B 0,C 180,E1 -20839.127,E2 -20839.127} C_VEL
LIN {X 0,Y 213.749,Z 557.845,A -85,B 0,C 180,E1 -20843.712,E2 -20843.712} C_VEL
LIN {X 0,Y 213.791,Z 557.85,A -85,B 0,C 180,E1 -20848.723,E2 -20848.723} C_VEL
LIN {X 0,Y 213.82,Z 557.836,A -85,B 0,C 180,E1 -20852.602,E2 -20852.602} C_VEL
LIN {X 0,Y 213.846,Z 557.834,A -85,B 0,C 180,E1 -20856.952,E2 -20856.952} C_VEL
LIN {X 0,Y 213.926,Z 557.827,A -85,B 0,C 180,E1 -20862.304,E2 -20862.304} C_VEL
LIN {X 0,Y 213.974,Z 557.83,A -85,B 0,C 180,E1 -20866.708,E2 -20866.708} C_VEL
LIN {X 0,Y 214.161,Z 557.788,A -85,B 0,C 180,E1 -20870.556,E2 -20870.556} C_VEL
LIN {X 0,Y 214.234,Z 557.796,A -85,B 0,C 180,E1 -20872.46,E2 -20872.46} C_VEL
LIN {X 0,Y 214.44,Z 557.758,A -85,B 0,C 180,E1 -20878.122,E2 -20878.122} C_VEL
LIN {X 0,Y 214.548,Z 557.761,A -85,B 0,C 180,E1 -20880,E2 -20880} C_VEL
LIN {X 0,Y 214.44,Z 557.765,A -85,B 0,C 180,E1 -20881.878,E2 -20881.878} C_VEL
LIN {X 0,Y 214.242,Z 557.797,A -85,B 0,C 180,E1 -20887.54,E2 -20887.54} C_VEL
LIN {X 0,Y 214.041,Z 557.81,A -85,B 0,C 180,E1 -20891.362,E2 -20891.362} C_VEL
LIN {X 0,Y 213.927,Z 557.824,A -85,B 0,C 180,E1 -20895.237,E2 -20895.237} C_VEL
LIN {X 0,Y 213.862,Z 557.846,A -85,B 0,C 180,E1 -20899.185,E2 -20899.185} C_VEL
LIN {X 0,Y 213.841,Z 557.843,A -85,B 0,C 180,E1 -20903.228,E2 -20903.228} C_VEL
LIN {X 0,Y 213.78,Z 557.845,A -85,B 0,C 180,E1 -20907.966,E2 -20907.966} C_VEL
LIN {X 0,Y 213.042,Z 557.947,A -85,B 0,C 180,E1 -20909.537,E2 -20909.537} C_VEL
LIN {X 0,Y 210.161,Z 558.302,A -85,B 0,C 180,E1 -20912.104,E2 -20912.104} C_VEL
LIN {X 0,Y 207.757,Z 558.595,A -85,B 0,C 180,E1 -20914.201,E2 -20914.201} C_VEL
LIN {X 0,Y 206.737,Z 558.703,A -85,B 0,C 180,E1 -20915.83,E2 -20915.83} C_VEL
LIN {X 0,Y 206.658,Z 558.711,A -85,B 0,C 180,E1 -20916.382,E2 -20916.382} C_VEL
LIN {X 0,Y 206.691,Z 558.736,A -85,B 0,C 180,E1 -20920.244,E2 -20920.244} C_VEL
LIN {X 0,Y 206.751,Z 558.922,A -85,B 0,C 180,E1 -20924.673,E2 -20924.673} C_VEL
LIN {X 0,Y 208.62,Z 565.807,A -85,B 0,C 180,E1 -20928.781,E2 -20928.781} C_VEL
LIN {X 0,Y 210.856,Z 570.096,A -85,B 0,C 180,E1 -20929.613,E2 -20929.613} C_VEL
LIN {X 0,Y 216.306,Z 580.127,A -85,B 0,C 180,E1 -20931.241,E2 -20931.241} C_VEL
LIN {X 0,Y 223.162,Z 594.658,A -85,B 0,C 180,E1 -20933.205,E2 -20933.205} C_VEL
LIN {X 0,Y 228.43,Z 607.686,A -85,B 0,C 180,E1 -20934.672,E2 -20934.672} C_VEL
LIN {X 0,Y 230.387,Z 622.834,A -85,B 0,C 180,E1 -20935.576,E2 -20935.576} C_VEL
LIN {X 0,Y 228.047,Z 674.687,A -85,B 0,C 180,E1 -20937.149,E2 -20937.149} C_VEL
LIN {X 0,Y 226.752,Z 687.73,A -85,B 0,C 180,E1 -20937.845,E2 -20937.845} C_VEL
LIN {X 0,Y 224.789,Z 700.194,A -85,B 0,C 180,E1 -20938.816,E2 -20938.816} C_VEL
LIN {X 0,Y 222.514,Z 712.402,A -85,B 0,C 180,E1 -20940.17,E2 -20940.17} C_VEL
LIN {X 0,Y 219.762,Z 723.961,A -85,B 0,C 180,E1 -20941.857,E2 -20941.857} C_VEL
LIN {X 0,Y 216.988,Z 734.374,A -85,B 0,C 180,E1 -20943.815,E2 -20943.815} C_VEL
LIN {X 0,Y 214.484,Z 742.892,A -85,B 0,C 180,E1 -20945.823,E2 -20945.823} C_VEL
LIN {X 0,Y 212.335,Z 750.162,A -85,B 0,C 180,E1 -20947.936,E2 -20947.936} C_VEL
LIN {X 0,Y 210.049,Z 757.28,A -85,B 0,C 180,E1 -20950.454,E2 -20950.454} C_VEL
LIN {X 0,Y 207.956,Z 763.701,A -85,B 0,C 180,E1 -20953.308,E2 -20953.308} C_VEL
LIN {X 0,Y 206.322,Z 768.804,A -85,B 0,C 180,E1 -20956.207,E2 -20956.207} C_VEL
LIN {X 0,Y 205.29,Z 772.778,A -85,B 0,C 180,E1 -20959.149,E2 -20959.149} C_VEL
LIN {X 0,Y 204.639,Z 775.717,A -85,B 0,C 180,E1 -20962.106,E2 -20962.106} C_VEL
LIN {X 0,Y 204.401,Z 777.113,A -85,B 0,C 180,E1 -20964.081,E2 -20964.081} C_VEL
LIN {X 0,Y 204.342,Z 778.721,A -85,B 0,C 180,E1 -20968.031,E2 -20968.031} C_VEL
LIN {X 0,Y 204.429,Z 778.935,A -85,B 0,C 180,E1 -20970.002,E2 -20970.002} C_VEL
LIN {X 0,Y 204.467,Z 778.712,A -85,B 0,C 180,E1 -20971.972,E2 -20971.972} C_VEL
LIN {X 0,Y 204.739,Z 778.037,A -85,B 0,C 180,E1 -20974.537,E2 -20974.537} C_VEL
LIN {X 0,Y 205.029,Z 781.177,A -85,B 0,C 180,E1 -20977.882,E2 -20977.882} C_VEL
LIN {X 0,Y 205.528,Z 782.317,A -85,B 0,C 180,E1 -20979.846,E2 -20979.846} C_VEL
LIN {X 0,Y 206.367,Z 782.981,A -85,B 0,C 180,E1 -20981.792,E2 -20981.792} C_VEL
LIN {X 0,Y 207.447,Z 783.169,A -85,B 0,C 180,E1 -20983.72,E2 -20983.72} C_VEL
LIN {X 0,Y 208.757,Z 782.807,A -85,B 0,C 180,E1 -20985.626,E2 -20985.626} C_VEL
LIN {X 0,Y 210.355,Z 781.909,A -85,B 0,C 180,E1 -20987.501,E2 -20987.501} C_VEL
LIN {X 0,Y 212.205,Z 780.531,A -85,B 0,C 180,E1 -20989.343,E2 -20989.343} C_VEL
LIN {X 0,Y 215.685,Z 777.48,A -85,B 0,C 180,E1 -20992.009,E2 -20992.009} C_VEL
LIN {X 0,Y 219.626,Z 773.184,A -85,B 0,C 180,E1 -20994.584,E2 -20994.584} C_VEL
LIN {X 0,Y 224.079,Z 767.307,A -85,B 0,C 180,E1 -20997.052,E2 -20997.052} C_VEL
LIN {X 0,Y 228.09,Z 761.307,A -85,B 0,C 180,E1 -20999.033,E2 -20999.033} C_VEL
LIN {X 0,Y 232.562,Z 753.76,A -85,B 0,C 180,E1 -21000.915,E2 -21000.915} C_VEL
LIN {X 0,Y 236.824,Z 745.413,A -85,B 0,C 180,E1 -21002.541,E2 -21002.541} C_VEL
LIN {X 0,Y 241.341,Z 735.073,A -85,B 0,C 180,E1 -21004.097,E2 -21004.097} C_VEL
LIN {X 0,Y 245.503,Z 723.19,A -85,B 0,C 180,E1 -21005.431,E2 -21005.431} C_VEL
LIN {X 0,Y 248.564,Z 711.901,A -85,B 0,C 180,E1 -21006.363,E2 -21006.363} C_VEL
LIN {X 0,Y 251.976,Z 695.1,A -85,B 0,C 180,E1 -21007.411,E2 -21007.411} C_VEL
LIN {X 0,Y 261.628,Z 650.056,A -85,B 0,C 180,E1 -21009.741,E2 -21009.741} C_VEL
LIN {X 0,Y 262.154,Z 647.405,A -85,B 0,C 180,E1 -21009.911,E2 -21009.911} C_VEL
LIN {X 0,Y 260.756,Z 646.652,A -85,B 0,C 180,E1 -21012.363,E2 -21012.363} C_VEL
LIN {X 0,Y 260.042,Z 647.225,A -85,B 0,C 180,E1 -21014.759,E2 -21014.759} C_VEL
LIN {X 0,Y 259.836,Z 649.383,A -85,B 0,C 180,E1 -21017.022,E2 -21017.022} C_VEL
LIN {X 0,Y 259.995,Z 652.294,A -85,B 0,C 180,E1 -21018.868,E2 -21018.868} C_VEL
LIN {X 0,Y 258.911,Z 662.907,A -85,B 0,C 180,E1 -21020.927,E2 -21020.927} C_VEL
LIN {X 0,Y 258.024,Z 674.068,A -85,B 0,C 180,E1 -21022.734,E2 -21022.734} C_VEL
LIN {X 0,Y 257.492,Z 681.434,A -85,B 0,C 180,E1 -21023.743,E2 -21023.743} C_VEL
LIN {X 0,Y 251.896,Z 709.143,A -85,B 0,C 180,E1 -21025.161,E2 -21025.161} C_VEL
LIN {X 0,Y 248.558,Z 721.649,A -85,B 0,C 180,E1 -21026.052,E2 -21026.052} C_VEL
LIN {X 0,Y 244.662,Z 732.52,A -85,B 0,C 180,E1 -21027.115,E2 -21027.115} C_VEL
LIN {X 0,Y 240.359,Z 742.494,A -85,B 0,C 180,E1 -21028.465,E2 -21028.465} C_VEL
LIN {X 0,Y 235.963,Z 750.928,A -85,B 0,C 180,E1 -21029.932,E2 -21029.932} C_VEL
LIN {X 0,Y 230.928,Z 759.316,A -85,B 0,C 180,E1 -21031.853,E2 -21031.853} C_VEL
LIN {X 0,Y 226.527,Z 765.473,A -85,B 0,C 180,E1 -21033.762,E2 -21033.762} C_VEL
LIN {X 0,Y 222.51,Z 770.474,A -85,B 0,C 180,E1 -21035.757,E2 -21035.757} C_VEL
LIN {X 0,Y 218.119,Z 775.061,A -85,B 0,C 180,E1 -21038.251,E2 -21038.251} C_VEL
LIN {X 0,Y 214.237,Z 778.164,A -85,B 0,C 180,E1 -21040.85,E2 -21040.85} C_VEL
LIN {X 0,Y 212.019,Z 779.594,A -85,B 0,C 180,E1 -21042.643,E2 -21042.643} C_VEL
LIN {X 0,Y 210.2,Z 780.472,A -85,B 0,C 180,E1 -21044.486,E2 -21044.486} C_VEL
LIN {X 0,Y 208.634,Z 780.78,A -85,B 0,C 180,E1 -21046.361,E2 -21046.361} C_VEL
LIN {X 0,Y 207.326,Z 780.571,A -85,B 0,C 180,E1 -21048.265,E2 -21048.265} C_VEL
LIN {X 0,Y 206.311,Z 779.868,A -85,B 0,C 180,E1 -21050.193,E2 -21050.193} C_VEL
LIN {X 0,Y 205.202,Z 777.677,A -85,B 0,C 180,E1 -21053.339,E2 -21053.339} C_VEL
LIN {X 0,Y 204.829,Z 774.639,A -85,B 0,C 180,E1 -21056.065,E2 -21056.065} C_VEL
LIN {X 0,Y 204.823,Z 769.894,A -85,B 0,C 180,E1 -21059.017,E2 -21059.017} C_VEL
LIN {X 0,Y 205.017,Z 764.739,A -85,B 0,C 180,E1 -21061.473,E2 -21061.473} C_VEL
LIN {X 0,Y 205.289,Z 759.642,A -85,B 0,C 180,E1 -21063.435,E2 -21063.435} C_VEL
LIN {X 0,Y 205.598,Z 751.593,A -85,B 0,C 180,E1 -21065.886,E2 -21065.886} C_VEL
LIN {X 0,Y 206.001,Z 743.395,A -85,B 0,C 180,E1 -21067.844,E2 -21067.844} C_VEL
LIN {X 0,Y 206.339,Z 735.751,A -85,B 0,C 180,E1 -21069.339,E2 -21069.339} C_VEL
LIN {X 0,Y 206.939,Z 724.96,A -85,B 0,C 180,E1 -21071.013,E2 -21071.013} C_VEL
LIN {X 0,Y 207.314,Z 714.431,A -85,B 0,C 180,E1 -21072.232,E2 -21072.232} C_VEL
LIN {X 0,Y 207.818,Z 700.927,A -85,B 0,C 180,E1 -21073.32,E2 -21073.32} C_VEL
LIN {X 0,Y 208.636,Z 656.439,A -85,B 0,C 180,E1 -21076.041,E2 -21076.041} C_VEL
LIN {X 0,Y 207.319,Z 634.775,A -85,B 0,C 180,E1 -21077.318,E2 -21077.318} C_VEL
LIN {X 0,Y 207.298,Z 632.242,A -85,B 0,C 180,E1 -21077.511,E2 -21077.511} C_VEL
LIN {X 0,Y 209.034,Z 611.985,A -85,B 0,C 180,E1 -21082.746,E2 -21082.746} C_VEL
LIN {X 0,Y 211.035,Z 592.36,A -85,B 0,C 180,E1 -21087.79,E2 -21087.79} C_VEL
LIN {X 0,Y 211.94,Z 584.39,A -85,B 0,C 180,E1 -21089.829,E2 -21089.829} C_VEL
LIN {X 0,Y 210.189,Z 575.114,A -85,B 0,C 180,E1 -21092.343,E2 -21092.343} C_VEL
LIN {X 0,Y 206.864,Z 558.933,A -85,B 0,C 180,E1 -21096.901,E2 -21096.901} C_VEL
LIN {X 0,Y 206.648,Z 558.687,A -85,B 0,C 180,E1 -21101.562,E2 -21101.562} C_VEL
LIN {X 0,Y 206.683,Z 558.707,A -85,B 0,C 180,E1 -21105.568,E2 -21105.568} C_VEL
LIN {X 0,Y 206.719,Z 558.977,A -85,B 0,C 180,E1 -21108.414,E2 -21108.414} C_VEL
LIN {X 0,Y 207.014,Z 560.065,A -85,B 0,C 180,E1 -21108.764,E2 -21108.764} C_VEL
LIN {X 0,Y 208.68,Z 562.791,A -85,B 0,C 180,E1 -21109.308,E2 -21109.308} C_VEL
LIN {X 0,Y 209.707,Z 564.171,A -85,B 0,C 180,E1 -21109.612,E2 -21109.612} C_VEL
LIN {X 0,Y 217.51,Z 576.617,A -85,B 0,C 180,E1 -21111.867,E2 -21111.867} C_VEL
LIN {X 0,Y 224.501,Z 590.664,A -85,B 0,C 180,E1 -21113.815,E2 -21113.815} C_VEL
LIN {X 0,Y 230.454,Z 604.827,A -85,B 0,C 180,E1 -21115.427,E2 -21115.427} C_VEL
LIN {X 0,Y 230.909,Z 606.041,A -85,B 0,C 180,E1 -21115.551,E2 -21115.551} C_VEL
LIN {X 0,Y 228.414,Z 663.252,A -85,B 0,C 180,E1 -21117.288,E2 -21117.288} C_VEL
LIN {X 0,Y 227.121,Z 676.522,A -85,B 0,C 180,E1 -21117.993,E2 -21117.993} C_VEL
LIN {X 0,Y 225.447,Z 689.318,A -85,B 0,C 180,E1 -21119.043,E2 -21119.043} C_VEL
LIN {X 0,Y 223.468,Z 700.607,A -85,B 0,C 180,E1 -21120.307,E2 -21120.307} C_VEL
LIN {X 0,Y 220.796,Z 712.241,A -85,B 0,C 180,E1 -21121.997,E2 -21121.997} C_VEL
LIN {X 0,Y 218.12,Z 722.687,A -85,B 0,C 180,E1 -21123.958,E2 -21123.958} C_VEL
LIN {X 0,Y 215.755,Z 731.253,A -85,B 0,C 180,E1 -21125.982,E2 -21125.982} C_VEL
LIN {X 0,Y 213.438,Z 739.073,A -85,B 0,C 180,E1 -21128.256,E2 -21128.256} C_VEL
LIN {X 0,Y 210.815,Z 746.753,A -85,B 0,C 180,E1 -21131.03,E2 -21131.03} C_VEL
LIN {X 0,Y 208.48,Z 753.801,A -85,B 0,C 180,E1 -21134.353,E2 -21134.353} C_VEL
LIN {X 0,Y 206.851,Z 758.494,A -85,B 0,C 180,E1 -21137.24,E2 -21137.24} C_VEL
LIN {X 0,Y 205.728,Z 762.077,A -85,B 0,C 180,E1 -21140.163,E2 -21140.163} C_VEL
LIN {X 0,Y 205.202,Z 763.927,A -85,B 0,C 180,E1 -21142.124,E2 -21142.124} C_VEL
LIN {X 0,Y 204.775,Z 765.519,A -85,B 0,C 180,E1 -21144.445,E2 -21144.445} C_VEL
LIN {X 0,Y 204.5,Z 766.916,A -85,B 0,C 180,E1 -21148.029,E2 -21148.029} C_VEL
LIN {X 0,Y 204.499,Z 767.144,A -85,B 0,C 180,E1 -21149.998,E2 -21149.998} C_VEL
LIN {X 0,Y 204.499,Z 766.951,A -85,B 0,C 180,E1 -21151.968,E2 -21151.968} C_VEL
LIN {X 0,Y 204.773,Z 765.603,A -85,B 0,C 180,E1 -21155.551,E2 -21155.551} C_VEL
LIN {X 0,Y 205.2,Z 764.046,A -85,B 0,C 180,E1 -21157.872,E2 -21157.872} C_VEL
LIN {X 0,Y 206.039,Z 761.177,A -85,B 0,C 180,E1 -21160.811,E2 -21160.811} C_VEL
LIN {X 0,Y 207.303,Z 757.284,A -85,B 0,C 180,E1 -21163.726,E2 -21163.726} C_VEL
LIN {X 0,Y 209.022,Z 752.264,A -85,B 0,C 180,E1 -21166.605,E2 -21166.605} C_VEL
LIN {X 0,Y 211.15,Z 745.94,A -85,B 0,C 180,E1 -21169.439,E2 -21169.439} C_VEL
LIN {X 0,Y 213.861,Z 738.019,A -85,B 0,C 180,E1 -21172.203,E2 -21172.203} C_VEL
LIN {X 0,Y 216.152,Z 730.125,A -85,B 0,C 180,E1 -21174.439,E2 -21174.439} C_VEL
LIN {X 0,Y 218.882,Z 720.101,A -85,B 0,C 180,E1 -21176.711,E2 -21176.711} C_VEL
LIN {X 0,Y 221.652,Z 709.007,A -85,B 0,C 180,E1 -21178.656,E2 -21178.656} C_VEL
LIN {X 0,Y 223.988,Z 698.123,A -85,B 0,C 180,E1 -21180.132,E2 -21180.132} C_VEL
LIN {X 0,Y 226.033,Z 686.085,A -85,B 0,C 180,E1 -21181.384,E2 -21181.384} C_VEL
LIN {X 0,Y 227.597,Z 673.954,A -85,B 0,C 180,E1 -21182.295,E2 -21182.295} C_VEL
LIN {X 0,Y 228.702,Z 660.743,A -85,B 0,C 180,E1 -21182.925,E2 -21182.925} C_VEL
LIN {X 0,Y 231.03,Z 606.184,A -85,B 0,C 180,E1 -21184.57,E2 -21184.57} C_VEL
LIN {X 0,Y 225.138,Z 592.107,A -85,B 0,C 180,E1 -21186.161,E2 -21186.161} C_VEL
LIN {X 0,Y 217.878,Z 577.229,A -85,B 0,C 180,E1 -21188.189,E2 -21188.189} C_VEL
LIN {X 0,Y 211.372,Z 566.81,A -85,B 0,C 180,E1 -21190.051,E2 -21190.051} C_VEL
LIN {X 0,Y 208.94,Z 563.087,A -85,B 0,C 180,E1 -21190.784,E2 -21190.784} C_VEL
LIN {X 0,Y 207.22,Z 560.728,A -85,B 0,C 180,E1 -21191.305,E2 -21191.305} C_VEL
